  MoveAbsJ [[102.02,-14.19,-142.83,-135.95,-26.88,37.39],[9E9,9E9,9E9,9E9,9E9,9E9]],speeddata0,DefaultBlend,tool0;
  MoveAbsJ [[101.51,-13.98,-141.84,-136.12,-26.41,37.13],[9E9,9E9,9E9,9E9,9E9,9E9]],speeddata0,DefaultBlend,tool0;
  MoveAbsJ [[100.99,-13.77,-140.85,-136.29,-25.94,36.87],[9E9,9E9,9E9,9E9,9E9,9E9]],speeddata0,DefaultBlend,tool0;
  MoveAbsJ [[100.48,-13.56,-139.86,-136.46,-25.48,36.61],[9E9,9E9,9E9,9E9,9E9,9E9]],speeddata0,DefaultBlend,tool0;
  MoveAbsJ [[99.97,-13.35,-138.87,-136.62,-25.01,36.35],[9E9,9E9,9E9,9E9,9E9,9E9]],speeddata0,DefaultBlend,tool0;
  MoveAbsJ [[99.46,-13.14,-137.88,-136.79,-24.54,36.09],[9E9,9E9,9E9,9E9,9E9,9E9]],speeddata0,DefaultBlend,tool0;
  MoveAbsJ [[98.95,-12.93,-136.89,-136.96,-24.08,35.83],[9E9,9E9,9E9,9E9,9E9,9E9]],speeddata0,DefaultBlend,tool0;
  MoveAbsJ [[98.43,-12.72,-135.89,-137.13,-23.61,35.57],[9E9,9E9,9E9,9E9,9E9,9E9]],speeddata0,DefaultBlend,tool0;
  MoveAbsJ [[97.92,-12.51,-134.90,-137.29,-23.14,35.31],[9E9,9E9,9E9,9E9,9E9,9E9]],speeddata0,DefaultBlend,tool0;
  MoveAbsJ [[97.41,-12.30,-133.91,-137.46,-22.68,35.05],[9E9,9E9,9E9,9E9,9E9,9E9]],speeddata0,DefaultBlend,tool0;
  MoveAbsJ [[96.90,-12.09,-132.92,-137.63,-22.21,34.79],[9E9,9E9,9E9,9E9,9E9,9E9]],speeddata0,DefaultBlend,tool0;
  MoveAbsJ [[96.39,-11.88,-131.93,-137.80,-21.74,34.53],[9E9,9E9,9E9,9E9,9E9,9E9]],speeddata0,DefaultBlend,tool0;
  MoveAbsJ [[95.87,-11.67,-130.94,-137.97,-21.28,34.27],[9E9,9E9,9E9,9E9,9E9,9E9]],speeddata0,DefaultBlend,tool0;
  MoveAbsJ [[95.36,-11.46,-129.95,-138.13,-20.81,34.01],[9E9,9E9,9E9,9E9,9E9,9E9]],speeddata0,DefaultBlend,tool0;
  MoveAbsJ [[94.85,-11.25,-128.96,-138.30,-20.34,33.75],[9E9,9E9,9E9,9E9,9E9,9E9]],speeddata0,DefaultBlend,tool0;
  MoveAbsJ [[94.34,-11.04,-127.96,-138.47,-19.88,33.49],[9E9,9E9,9E9,9E9,9E9,9E9]],speeddata0,DefaultBlend,tool0;
  MoveAbsJ [[93.83,-10.83,-126.97,-138.64,-19.41,33.23],[9E9,9E9,9E9,9E9,9E9,9E9]],speeddata0,DefaultBlend,tool0;
  MoveAbsJ [[93.31,-10.63,-125.98,-138.80,-18.94,32.97],[9E9,9E9,9E9,9E9,9E9,9E9]],speeddata0,DefaultBlend,tool0;
  MoveAbsJ [[92.80,-10.42,-124.99,-138.97,-18.48,32.71],[9E9,9E9,9E9,9E9,9E9,9E9]],speeddata0,DefaultBlend,tool0;
  MoveAbsJ [[92.29,-10.21,-124.00,-139.14,-18.01,32.45],[9E9,9E9,9E9,9E9,9E9,9E9]],speeddata0,DefaultBlend,tool0;
  MoveAbsJ [[91.78,-10.00,-123.01,-139.31,-17.54,32.19],[9E9,9E9,9E9,9E9,9E9,9E9]],speeddata0,DefaultBlend,tool0;
  MoveAbsJ [[91.27,-9.79,-122.02,-139.47,-17.08,31.93],[9E9,9E9,9E9,9E9,9E9,9E9]],speeddata0,DefaultBlend,tool0;
  MoveAbsJ [[90.75,-9.58,-121.02,-139.64,-16.61,31.67],[9E9,9E9,9E9,9E9,9E9,9E9]],speeddata0,DefaultBlend,tool0;
  MoveAbsJ [[90.24,-9.37,-120.03,-139.81,-16.14,31.41],[9E9,9E9,9E9,9E9,9E9,9E9]],speeddata0,DefaultBlend,tool0;
  MoveAbsJ [[89.73,-9.16,-119.04,-139.98,-15.68,31.15],[9E9,9E9,9E9,9E9,9E9,9E9]],speeddata0,DefaultBlend,tool0;
  MoveAbsJ [[89.22,-8.95,-118.05,-140.14,-15.21,30.89],[9E9,9E9,9E9,9E9,9E9,9E9]],speeddata0,DefaultBlend,tool0;
  MoveAbsJ [[88.71,-8.74,-117.06,-140.31,-14.74,30.63],[9E9,9E9,9E9,9E9,9E9,9E9]],speeddata0,DefaultBlend,tool0;
  MoveAbsJ [[88.19,-8.53,-116.07,-140.48,-14.28,30.36],[9E9,9E9,9E9,9E9,9E9,9E9]],speeddata0,DefaultBlend,tool0;
  MoveAbsJ [[87.68,-8.32,-115.08,-140.65,-13.81,30.10],[9E9,9E9,9E9,9E9,9E9,9E9]],speeddata0,DefaultBlend,tool0;
  MoveAbsJ [[87.17,-8.11,-114.08,-140.82,-13.34,29.84],[9E9,9E9,9E9,9E9,9E9,9E9]],speeddata0,DefaultBlend,tool0;
  MoveAbsJ [[86.66,-7.90,-113.09,-140.98,-12.88,29.58],[9E9,9E9,9E9,9E9,9E9,9E9]],speeddata0,DefaultBlend,tool0;
  MoveAbsJ [[86.15,-7.69,-112.10,-141.15,-12.41,29.32],[9E9,9E9,9E9,9E9,9E9,9E9]],speeddata0,DefaultBlend,tool0;
  MoveAbsJ [[85.63,-7.48,-111.11,-141.32,-11.94,29.06],[9E9,9E9,9E9,9E9,9E9,9E9]],speeddata0,DefaultBlend,tool0;
  MoveAbsJ [[85.12,-7.27,-110.12,-141.49,-11.48,28.80],[9E9,9E9,9E9,9E9,9E9,9E9]],speeddata0,DefaultBlend,tool0;
  MoveAbsJ [[84.61,-7.06,-109.13,-141.65,-11.01,28.54],[9E9,9E9,9E9,9E9,9E9,9E9]],speeddata0,DefaultBlend,tool0;
  MoveAbsJ [[84.10,-6.85,-108.14,-141.82,-10.54,28.28],[9E9,9E9,9E9,9E9,9E9,9E9]],speeddata0,DefaultBlend,tool0;
  MoveAbsJ [[83.59,-6.64,-107.15,-141.99,-10.08,28.02],[9E9,9E9,9E9,9E9,9E9,9E9]],speeddata0,DefaultBlend,tool0;
  MoveAbsJ [[83.07,-6.43,-106.15,-142.16,-9.61,27.76],[9E9,9E9,9E9,9E9,9E9,9E9]],speeddata0,DefaultBlend,tool0;
  MoveAbsJ [[82.56,-6.22,-105.16,-142.32,-9.14,27.50],[9E9,9E9,9E9,9E9,9E9,9E9]],speeddata0,DefaultBlend,tool0;
  MoveAbsJ [[82.05,-6.01,-104.17,-142.49,-8.68,27.24],[9E9,9E9,9E9,9E9,9E9,9E9]],speeddata0,DefaultBlend,tool0;
  MoveAbsJ [[81.54,-5.80,-103.18,-142.66,-8.21,26.98],[9E9,9E9,9E9,9E9,9E9,9E9]],speeddata0,DefaultBlend,tool0;
  MoveAbsJ [[81.03,-5.59,-102.19,-142.83,-7.74,26.72],[9E9,9E9,9E9,9E9,9E9,9E9]],speeddata0,DefaultBlend,tool0;
  MoveAbsJ [[80.51,-5.38,-101.20,-142.99,-7.28,26.46],[9E9,9E9,9E9,9E9,9E9,9E9]],speeddata0,DefaultBlend,tool0;
  MoveAbsJ [[80.00,-5.17,-100.21,-143.16,-6.81,26.20],[9E9,9E9,9E9,9E9,9E9,9E9]],speeddata0,DefaultBlend,tool0;
  MoveAbsJ [[79.49,-4.96,-99.21,-143.33,-6.34,25.94],[9E9,9E9,9E9,9E9,9E9,9E9]],speeddata0,DefaultBlend,tool0;
  MoveAbsJ [[78.98,-4.75,-98.22,-143.50,-5.88,25.68],[9E9,9E9,9E9,9E9,9E9,9E9]],speeddata0,DefaultBlend,tool0;
  MoveAbsJ [[78.46,-4.54,-97.23,-143.67,-5.41,25.42],[9E9,9E9,9E9,9E9,9E9,9E9]],speeddata0,DefaultBlend,tool0;
  MoveAbsJ [[77.95,-4.33,-96.24,-143.83,-4.94,25.16],[9E9,9E9,9E9,9E9,9E9,9E9]],speeddata0,DefaultBlend,tool0;
  MoveAbsJ [[77.44,-4.13,-95.25,-144.00,-4.48,24.90],[9E9,9E9,9E9,9E9,9E9,9E9]],speeddata0,DefaultBlend,tool0;
  MoveAbsJ [[76.93,-3.92,-94.26,-144.17,-4.01,24.64],[9E9,9E9,9E9,9E9,9E9,9E9]],speeddata0,DefaultBlend,tool0;
  MoveAbsJ [[76.42,-3.71,-93.27,-144.34,-3.54,24.38],[9E9,9E9,9E9,9E9,9E9,9E9]],speeddata0,DefaultBlend,tool0;
  MoveAbsJ [[75.90,-3.50,-92.28,-144.50,-3.08,24.12],[9E9,9E9,9E9,9E9,9E9,9E9]],speeddata0,DefaultBlend,tool0;
  MoveAbsJ [[75.39,-3.29,-91.28,-144.67,-2.61,23.86],[9E9,9E9,9E9,9E9,9E9,9E9]],speeddata0,DefaultBlend,tool0;
  MoveAbsJ [[74.88,-3.08,-90.29,-144.84,-2.14,23.60],[9E9,9E9,9E9,9E9,9E9,9E9]],speeddata0,DefaultBlend,tool0;
  MoveAbsJ [[74.37,-2.87,-89.30,-145.01,-1.68,23.34],[9E9,9E9,9E9,9E9,9E9,9E9]],speeddata0,DefaultBlend,tool0;
  MoveAbsJ [[73.86,-2.66,-88.31,-145.17,-1.21,23.08],[9E9,9E9,9E9,9E9,9E9,9E9]],speeddata0,DefaultBlend,tool0;
  MoveAbsJ [[73.34,-2.45,-87.32,-145.34,-0.74,22.82],[9E9,9E9,9E9,9E9,9E9,9E9]],speeddata0,DefaultBlend,tool0;
  MoveAbsJ [[72.83,-2.24,-86.33,-145.51,-0.28,22.56],[9E9,9E9,9E9,9E9,9E9,9E9]],speeddata0,DefaultBlend,tool0;
  MoveAbsJ [[72.32,-2.03,-85.34,-145.68,0.19,22.30],[9E9,9E9,9E9,9E9,9E9,9E9]],speeddata0,DefaultBlend,tool0;
  MoveAbsJ [[71.81,-1.82,-84.34,-145.85,0.66,22.04],[9E9,9E9,9E9,9E9,9E9,9E9]],speeddata0,DefaultBlend,tool0;
  MoveAbsJ [[71.30,-1.61,-83.35,-146.01,1.12,21.78],[9E9,9E9,9E9,9E9,9E9,9E9]],speeddata0,DefaultBlend,tool0;
  MoveAbsJ [[70.78,-1.40,-82.36,-146.18,1.59,21.52],[9E9,9E9,9E9,9E9,9E9,9E9]],speeddata0,DefaultBlend,tool0;
  MoveAbsJ [[70.27,-1.19,-81.37,-146.35,2.06,21.26],[9E9,9E9,9E9,9E9,9E9,9E9]],speeddata0,DefaultBlend,tool0;
  MoveAbsJ [[69.76,-0.98,-80.38,-146.52,2.52,21.00],[9E9,9E9,9E9,9E9,9E9,9E9]],speeddata0,DefaultBlend,tool0;
  MoveAbsJ [[69.25,-0.77,-79.39,-146.68,2.99,20.74],[9E9,9E9,9E9,9E9,9E9,9E9]],speeddata0,DefaultBlend,tool0;
  MoveAbsJ [[68.74,-0.56,-78.40,-146.85,3.46,20.48],[9E9,9E9,9E9,9E9,9E9,9E9]],speeddata0,DefaultBlend,tool0;
  MoveAbsJ [[68.22,-0.35,-77.40,-147.02,3.92,20.22],[9E9,9E9,9E9,9E9,9E9,9E9]],speeddata0,DefaultBlend,tool0;
  MoveAbsJ [[67.71,-0.14,-76.41,-147.19,4.39,19.96],[9E9,9E9,9E9,9E9,9E9,9E9]],speeddata0,DefaultBlend,tool0;
  MoveAbsJ [[67.20,0.07,-75.42,-147.35,4.86,19.70],[9E9,9E9,9E9,9E9,9E9,9E9]],speeddata0,DefaultBlend,tool0;
  MoveAbsJ [[66.69,0.28,-74.43,-147.52,5.32,19.43],[9E9,9E9,9E9,9E9,9E9,9E9]],speeddata0,DefaultBlend,tool0;
  MoveAbsJ [[66.18,0.49,-73.44,-147.69,5.79,19.17],[9E9,9E9,9E9,9E9,9E9,9E9]],speeddata0,DefaultBlend,tool0;
  MoveAbsJ [[65.66,0.70,-72.45,-147.86,6.26,18.91],[9E9,9E9,9E9,9E9,9E9,9E9]],speeddata0,DefaultBlend,tool0;
  MoveAbsJ [[65.15,0.91,-71.46,-148.02,6.72,18.65],[9E9,9E9,9E9,9E9,9E9,9E9]],speeddata0,DefaultBlend,tool0;
  MoveAbsJ [[64.64,1.12,-70.47,-148.19,7.19,18.39],[9E9,9E9,9E9,9E9,9E9,9E9]],speeddata0,DefaultBlend,tool0;
  MoveAbsJ [[64.13,1.33,-69.47,-148.36,7.66,18.13],[9E9,9E9,9E9,9E9,9E9,9E9]],speeddata0,DefaultBlend,tool0;
  MoveAbsJ [[63.62,1.54,-68.48,-148.53,8.12,17.87],[9E9,9E9,9E9,9E9,9E9,9E9]],speeddata0,DefaultBlend,tool0;
  MoveAbsJ [[63.10,1.75,-67.49,-148.70,8.59,17.61],[9E9,9E9,9E9,9E9,9E9,9E9]],speeddata0,DefaultBlend,tool0;
  MoveAbsJ [[62.59,1.96,-66.50,-148.86,9.06,17.35],[9E9,9E9,9E9,9E9,9E9,9E9]],speeddata0,DefaultBlend,tool0;
  MoveAbsJ [[62.08,2.17,-65.51,-149.03,9.52,17.09],[9E9,9E9,9E9,9E9,9E9,9E9]],speeddata0,DefaultBlend,tool0;
  MoveAbsJ [[61.57,2.37,-64.52,-149.20,9.99,16.83],[9E9,9E9,9E9,9E9,9E9,9E9]],speeddata0,DefaultBlend,tool0;
  MoveAbsJ [[61.06,2.58,-63.53,-149.37,10.46,16.57],[9E9,9E9,9E9,9E9,9E9,9E9]],speeddata0,DefaultBlend,tool0;
  MoveAbsJ [[60.54,2.79,-62.53,-149.53,10.92,16.31],[9E9,9E9,9E9,9E9,9E9,9E9]],speeddata0,DefaultBlend,tool0;
  MoveAbsJ [[60.03,3.00,-61.54,-149.70,11.39,16.05],[9E9,9E9,9E9,9E9,9E9,9E9]],speeddata0,DefaultBlend,tool0;
  MoveAbsJ [[59.52,3.21,-60.55,-149.87,11.86,15.79],[9E9,9E9,9E9,9E9,9E9,9E9]],speeddata0,DefaultBlend,tool0;
  MoveAbsJ [[59.01,3.42,-59.56,-150.04,12.32,15.53],[9E9,9E9,9E9,9E9,9E9,9E9]],speeddata0,DefaultBlend,tool0;
  MoveAbsJ [[58.50,3.63,-58.57,-150.20,12.79,15.27],[9E9,9E9,9E9,9E9,9E9,9E9]],speeddata0,DefaultBlend,tool0;
  MoveAbsJ [[57.98,3.84,-57.58,-150.37,13.26,15.01],[9E9,9E9,9E9,9E9,9E9,9E9]],speeddata0,DefaultBlend,tool0;
  MoveAbsJ [[57.47,4.05,-56.59,-150.54,13.72,14.75],[9E9,9E9,9E9,9E9,9E9,9E9]],speeddata0,DefaultBlend,tool0;
  MoveAbsJ [[56.96,4.26,-55.59,-150.71,14.19,14.49],[9E9,9E9,9E9,9E9,9E9,9E9]],speeddata0,DefaultBlend,tool0;
  MoveAbsJ [[56.45,4.47,-54.60,-150.87,14.66,14.23],[9E9,9E9,9E9,9E9,9E9,9E9]],speeddata0,DefaultBlend,tool0;
  MoveAbsJ [[55.94,4.68,-53.61,-151.04,15.12,13.97],[9E9,9E9,9E9,9E9,9E9,9E9]],speeddata0,DefaultBlend,tool0;
  MoveAbsJ [[55.42,4.89,-52.62,-151.21,15.59,13.71],[9E9,9E9,9E9,9E9,9E9,9E9]],speeddata0,DefaultBlend,tool0;
  MoveAbsJ [[54.91,5.10,-51.63,-151.38,16.06,13.45],[9E9,9E9,9E9,9E9,9E9,9E9]],speeddata0,DefaultBlend,tool0;
  MoveAbsJ [[54.40,5.31,-50.64,-151.55,16.52,13.19],[9E9,9E9,9E9,9E9,9E9,9E9]],speeddata0,DefaultBlend,tool0;
  MoveAbsJ [[53.89,5.52,-49.65,-151.71,16.99,12.93],[9E9,9E9,9E9,9E9,9E9,9E9]],speeddata0,DefaultBlend,tool0;
  MoveAbsJ [[53.38,5.73,-48.66,-151.88,17.46,12.67],[9E9,9E9,9E9,9E9,9E9,9E9]],speeddata0,DefaultBlend,tool0;
  MoveAbsJ [[52.86,5.94,-47.66,-152.05,17.92,12.41],[9E9,9E9,9E9,9E9,9E9,9E9]],speeddata0,DefaultBlend,tool0;
  MoveAbsJ [[52.35,6.15,-46.67,-152.22,18.39,12.15],[9E9,9E9,9E9,9E9,9E9,9E9]],speeddata0,DefaultBlend,tool0;
  MoveAbsJ [[51.84,6.36,-45.68,-152.38,18.85,11.89],[9E9,9E9,9E9,9E9,9E9,9E9]],speeddata0,DefaultBlend,tool0;
  MoveAbsJ [[51.33,6.57,-44.69,-152.55,19.32,11.63],[9E9,9E9,9E9,9E9,9E9,9E9]],speeddata0,DefaultBlend,tool0;
  MoveAbsJ [[50.82,6.78,-43.70,-152.72,19.79,11.37],[9E9,9E9,9E9,9E9,9E9,9E9]],speeddata0,DefaultBlend,tool0;
  MoveAbsJ [[50.30,6.99,-42.71,-152.89,20.25,11.11],[9E9,9E9,9E9,9E9,9E9,9E9]],speeddata0,DefaultBlend,tool0;
  MoveAbsJ [[49.79,7.20,-41.72,-153.05,20.72,10.85],[9E9,9E9,9E9,9E9,9E9,9E9]],speeddata0,DefaultBlend,tool0;
  MoveAbsJ [[49.28,7.41,-40.72,-153.22,21.19,10.59],[9E9,9E9,9E9,9E9,9E9,9E9]],speeddata0,DefaultBlend,tool0;
  MoveAbsJ [[48.77,7.62,-39.73,-153.39,21.65,10.33],[9E9,9E9,9E9,9E9,9E9,9E9]],speeddata0,DefaultBlend,tool0;
  MoveAbsJ [[48.26,7.83,-38.74,-153.56,22.12,10.07],[9E9,9E9,9E9,9E9,9E9,9E9]],speeddata0,DefaultBlend,tool0;
  MoveAbsJ [[47.74,8.04,-37.75,-153.73,22.59,9.81],[9E9,9E9,9E9,9E9,9E9,9E9]],speeddata0,DefaultBlend,tool0;
  MoveAbsJ [[47.23,8.25,-36.76,-153.89,23.05,9.55],[9E9,9E9,9E9,9E9,9E9,9E9]],speeddata0,DefaultBlend,tool0;
  MoveAbsJ [[46.72,8.46,-35.77,-154.06,23.52,9.29],[9E9,9E9,9E9,9E9,9E9,9E9]],speeddata0,DefaultBlend,tool0;
  MoveAbsJ [[46.21,8.66,-34.78,-154.23,23.99,9.03],[9E9,9E9,9E9,9E9,9E9,9E9]],speeddata0,DefaultBlend,tool0;
  MoveAbsJ [[45.69,8.87,-33.79,-154.40,24.45,8.77],[9E9,9E9,9E9,9E9,9E9,9E9]],speeddata0,DefaultBlend,tool0;
  MoveAbsJ [[45.18,9.08,-32.79,-154.56,24.92,8.50],[9E9,9E9,9E9,9E9,9E9,9E9]],speeddata0,DefaultBlend,tool0;
  MoveAbsJ [[44.67,9.29,-31.80,-154.73,25.39,8.24],[9E9,9E9,9E9,9E9,9E9,9E9]],speeddata0,DefaultBlend,tool0;
  MoveAbsJ [[44.16,9.50,-30.81,-154.90,25.85,7.98],[9E9,9E9,9E9,9E9,9E9,9E9]],speeddata0,DefaultBlend,tool0;
  MoveAbsJ [[43.65,9.71,-29.82,-155.07,26.32,7.72],[9E9,9E9,9E9,9E9,9E9,9E9]],speeddata0,DefaultBlend,tool0;
  MoveAbsJ [[43.13,9.92,-28.83,-155.23,26.79,7.46],[9E9,9E9,9E9,9E9,9E9,9E9]],speeddata0,DefaultBlend,tool0;
  MoveAbsJ [[42.62,10.13,-27.84,-155.40,27.25,7.20],[9E9,9E9,9E9,9E9,9E9,9E9]],speeddata0,DefaultBlend,tool0;
  MoveAbsJ [[42.11,10.34,-26.85,-155.57,27.72,6.94],[9E9,9E9,9E9,9E9,9E9,9E9]],speeddata0,DefaultBlend,tool0;
  MoveAbsJ [[41.60,10.55,-25.85,-155.74,28.19,6.68],[9E9,9E9,9E9,9E9,9E9,9E9]],speeddata0,DefaultBlend,tool0;
  MoveAbsJ [[41.09,10.76,-24.86,-155.90,28.65,6.42],[9E9,9E9,9E9,9E9,9E9,9E9]],speeddata0,DefaultBlend,tool0;
  MoveAbsJ [[40.57,10.97,-23.87,-156.07,29.12,6.16],[9E9,9E9,9E9,9E9,9E9,9E9]],speeddata0,DefaultBlend,tool0;
  MoveAbsJ [[40.06,11.18,-22.88,-156.24,29.59,5.90],[9E9,9E9,9E9,9E9,9E9,9E9]],speeddata0,DefaultBlend,tool0;
  MoveAbsJ [[39.55,11.39,-21.89,-156.41,30.05,5.64],[9E9,9E9,9E9,9E9,9E9,9E9]],speeddata0,DefaultBlend,tool0;
  MoveAbsJ [[39.04,11.60,-20.90,-156.58,30.52,5.38],[9E9,9E9,9E9,9E9,9E9,9E9]],speeddata0,DefaultBlend,tool0;
  MoveAbsJ [[38.53,11.81,-19.91,-156.74,30.99,5.12],[9E9,9E9,9E9,9E9,9E9,9E9]],speeddata0,DefaultBlend,tool0;
  MoveAbsJ [[38.01,12.02,-18.91,-156.91,31.45,4.86],[9E9,9E9,9E9,9E9,9E9,9E9]],speeddata0,DefaultBlend,tool0;
  MoveAbsJ [[37.50,12.23,-17.92,-157.08,31.92,4.60],[9E9,9E9,9E9,9E9,9E9,9E9]],speeddata0,DefaultBlend,tool0;
  MoveAbsJ [[36.99,12.44,-16.93,-157.25,32.39,4.34],[9E9,9E9,9E9,9E9,9E9,9E9]],speeddata0,DefaultBlend,tool0;
  MoveAbsJ [[36.48,12.65,-15.94,-157.41,32.85,4.08],[9E9,9E9,9E9,9E9,9E9,9E9]],speeddata0,DefaultBlend,tool0;
  MoveAbsJ [[35.97,12.86,-14.95,-157.58,33.32,3.82],[9E9,9E9,9E9,9E9,9E9,9E9]],speeddata0,DefaultBlend,tool0;
  MoveAbsJ [[35.45,13.07,-13.96,-157.75,33.79,3.56],[9E9,9E9,9E9,9E9,9E9,9E9]],speeddata0,DefaultBlend,tool0;
  MoveAbsJ [[34.94,13.28,-12.97,-157.92,34.25,3.30],[9E9,9E9,9E9,9E9,9E9,9E9]],speeddata0,DefaultBlend,tool0;
  MoveAbsJ [[34.43,13.49,-11.98,-158.08,34.72,3.04],[9E9,9E9,9E9,9E9,9E9,9E9]],speeddata0,DefaultBlend,tool0;
  MoveAbsJ [[33.92,13.70,-10.98,-158.25,35.19,2.78],[9E9,9E9,9E9,9E9,9E9,9E9]],speeddata0,DefaultBlend,tool0;
  MoveAbsJ [[33.41,13.91,-9.99,-158.42,35.65,2.52],[9E9,9E9,9E9,9E9,9E9,9E9]],speeddata0,DefaultBlend,tool0;
  MoveAbsJ [[32.89,14.12,-9.00,-158.59,36.12,2.26],[9E9,9E9,9E9,9E9,9E9,9E9]],speeddata0,DefaultBlend,tool0;
  MoveAbsJ [[32.38,14.33,-8.01,-158.75,36.59,2.00],[9E9,9E9,9E9,9E9,9E9,9E9]],speeddata0,DefaultBlend,tool0;
  MoveAbsJ [[31.87,14.54,-7.02,-158.92,37.05,1.74],[9E9,9E9,9E9,9E9,9E9,9E9]],speeddata0,DefaultBlend,tool0;
  MoveAbsJ [[31.36,14.75,-6.03,-159.09,37.52,1.48],[9E9,9E9,9E9,9E9,9E9,9E9]],speeddata0,DefaultBlend,tool0;
  MoveAbsJ [[30.85,14.96,-5.04,-159.26,37.99,1.22],[9E9,9E9,9E9,9E9,9E9,9E9]],speeddata0,DefaultBlend,tool0;
  MoveAbsJ [[30.33,15.16,-4.04,-159.43,38.45,0.96],[9E9,9E9,9E9,9E9,9E9,9E9]],speeddata0,DefaultBlend,tool0;
  MoveAbsJ [[29.82,15.37,-3.05,-159.59,38.92,0.70],[9E9,9E9,9E9,9E9,9E9,9E9]],speeddata0,DefaultBlend,tool0;
  MoveAbsJ [[29.31,15.58,-2.06,-159.76,39.39,0.44],[9E9,9E9,9E9,9E9,9E9,9E9]],speeddata0,DefaultBlend,tool0;
  MoveAbsJ [[28.80,15.79,-1.07,-159.93,39.85,0.18],[9E9,9E9,9E9,9E9,9E9,9E9]],speeddata0,DefaultBlend,tool0;
  MoveAbsJ [[28.29,16.00,-0.08,-160.10,40.32,-0.08],[9E9,9E9,9E9,9E9,9E9,9E9]],speeddata0,DefaultBlend,tool0;
  MoveAbsJ [[27.77,16.21,0.91,-160.26,40.79,-0.34],[9E9,9E9,9E9,9E9,9E9,9E9]],speeddata0,DefaultBlend,tool0;
  MoveAbsJ [[27.26,16.42,1.90,-160.43,41.25,-0.60],[9E9,9E9,9E9,9E9,9E9,9E9]],speeddata0,DefaultBlend,tool0;
  MoveAbsJ [[26.75,16.63,2.90,-160.60,41.72,-0.86],[9E9,9E9,9E9,9E9,9E9,9E9]],speeddata0,DefaultBlend,tool0;
  MoveAbsJ [[26.24,16.84,3.89,-160.77,42.19,-1.12],[9E9,9E9,9E9,9E9,9E9,9E9]],speeddata0,DefaultBlend,tool0;
  MoveAbsJ [[25.73,17.05,4.88,-160.93,42.65,-1.38],[9E9,9E9,9E9,9E9,9E9,9E9]],speeddata0,DefaultBlend,tool0;
  MoveAbsJ [[25.21,17.26,5.87,-161.10,43.12,-1.64],[9E9,9E9,9E9,9E9,9E9,9E9]],speeddata0,DefaultBlend,tool0;
  MoveAbsJ [[24.70,17.47,6.86,-161.27,43.59,-1.90],[9E9,9E9,9E9,9E9,9E9,9E9]],speeddata0,DefaultBlend,tool0;
  MoveAbsJ [[24.19,17.68,7.85,-161.44,44.05,-2.16],[9E9,9E9,9E9,9E9,9E9,9E9]],speeddata0,DefaultBlend,tool0;
  MoveAbsJ [[23.68,17.89,8.84,-161.60,44.52,-2.42],[9E9,9E9,9E9,9E9,9E9,9E9]],speeddata0,DefaultBlend,tool0;
  MoveAbsJ [[23.17,18.10,9.83,-161.77,44.99,-2.69],[9E9,9E9,9E9,9E9,9E9,9E9]],speeddata0,DefaultBlend,tool0;
  MoveAbsJ [[22.65,18.31,10.83,-161.94,45.45,-2.95],[9E9,9E9,9E9,9E9,9E9,9E9]],speeddata0,DefaultBlend,tool0;
  MoveAbsJ [[22.14,18.52,11.82,-162.11,45.92,-3.21],[9E9,9E9,9E9,9E9,9E9,9E9]],speeddata0,DefaultBlend,tool0;
  MoveAbsJ [[21.63,18.73,12.81,-162.28,46.39,-3.47],[9E9,9E9,9E9,9E9,9E9,9E9]],speeddata0,DefaultBlend,tool0;
  MoveAbsJ [[21.12,18.94,13.80,-162.44,46.85,-3.73],[9E9,9E9,9E9,9E9,9E9,9E9]],speeddata0,DefaultBlend,tool0;
  MoveAbsJ [[20.61,19.15,14.79,-162.61,47.32,-3.99],[9E9,9E9,9E9,9E9,9E9,9E9]],speeddata0,DefaultBlend,tool0;
  MoveAbsJ [[20.09,19.36,15.78,-162.78,47.79,-4.25],[9E9,9E9,9E9,9E9,9E9,9E9]],speeddata0,DefaultBlend,tool0;
  MoveAbsJ [[19.58,19.57,16.77,-162.95,48.25,-4.51],[9E9,9E9,9E9,9E9,9E9,9E9]],speeddata0,DefaultBlend,tool0;
  MoveAbsJ [[19.07,19.78,17.77,-163.11,48.72,-4.77],[9E9,9E9,9E9,9E9,9E9,9E9]],speeddata0,DefaultBlend,tool0;
  MoveAbsJ [[18.56,19.99,18.76,-163.28,49.19,-5.03],[9E9,9E9,9E9,9E9,9E9,9E9]],speeddata0,DefaultBlend,tool0;
  MoveAbsJ [[18.05,20.20,19.75,-163.45,49.65,-5.29],[9E9,9E9,9E9,9E9,9E9,9E9]],speeddata0,DefaultBlend,tool0;
  MoveAbsJ [[17.53,20.41,20.74,-163.62,50.12,-5.55],[9E9,9E9,9E9,9E9,9E9,9E9]],speeddata0,DefaultBlend,tool0;
  MoveAbsJ [[17.02,20.62,21.73,-163.78,50.59,-5.81],[9E9,9E9,9E9,9E9,9E9,9E9]],speeddata0,DefaultBlend,tool0;
  MoveAbsJ [[16.51,20.83,22.72,-163.95,51.05,-6.07],[9E9,9E9,9E9,9E9,9E9,9E9]],speeddata0,DefaultBlend,tool0;
  MoveAbsJ [[16.00,21.04,23.71,-164.12,51.52,-6.33],[9E9,9E9,9E9,9E9,9E9,9E9]],speeddata0,DefaultBlend,tool0;
  MoveAbsJ [[15.49,21.25,24.70,-164.29,51.99,-6.59],[9E9,9E9,9E9,9E9,9E9,9E9]],speeddata0,DefaultBlend,tool0;
  MoveAbsJ [[14.97,21.46,25.70,-164.46,52.45,-6.85],[9E9,9E9,9E9,9E9,9E9,9E9]],speeddata0,DefaultBlend,tool0;
  MoveAbsJ [[14.46,21.66,26.69,-164.62,52.92,-7.11],[9E9,9E9,9E9,9E9,9E9,9E9]],speeddata0,DefaultBlend,tool0;
  MoveAbsJ [[13.95,21.87,27.68,-164.79,53.39,-7.37],[9E9,9E9,9E9,9E9,9E9,9E9]],speeddata0,DefaultBlend,tool0;
  MoveAbsJ [[13.44,22.08,28.67,-164.96,53.85,-7.63],[9E9,9E9,9E9,9E9,9E9,9E9]],speeddata0,DefaultBlend,tool0;
  MoveAbsJ [[12.93,22.29,29.66,-165.13,54.32,-7.89],[9E9,9E9,9E9,9E9,9E9,9E9]],speeddata0,DefaultBlend,tool0;
  MoveAbsJ [[12.41,22.50,30.65,-165.29,54.79,-8.15],[9E9,9E9,9E9,9E9,9E9,9E9]],speeddata0,DefaultBlend,tool0;
  MoveAbsJ [[11.90,22.71,31.64,-165.46,55.25,-8.41],[9E9,9E9,9E9,9E9,9E9,9E9]],speeddata0,FinePoint,tool0;
  TPWrite "Action 39 LinearMovement.";
  MoveAbsJ [[11.90,22.71,31.64,-165.46,55.25,-8.41],[9E9,9E9,9E9,9E9,9E9,9E9]],speeddata0,DefaultBlend,tool0;
  MoveAbsJ [[11.88,22.74,31.53,-165.47,55.15,-8.42],[9E9,9E9,9E9,9E9,9E9,9E9]],speeddata0,DefaultBlend,tool0;
  MoveAbsJ [[12.53,23.48,31.49,-164.82,55.92,-8.64],[9E9,9E9,9E9,9E9,9E9,9E9]],speeddata0,DefaultBlend,tool0;
  MoveAbsJ [[13.19,24.23,31.43,-164.16,56.68,-8.86],[9E9,9E9,9E9,9E9,9E9,9E9]],speeddata0,DefaultBlend,tool0;
  MoveAbsJ [[13.85,24.99,31.35,-163.51,57.44,-9.05],[9E9,9E9,9E9,9E9,9E9,9E9]],speeddata0,DefaultBlend,tool0;
  MoveAbsJ [[14.50,25.77,31.24,-162.86,58.19,-9.23],[9E9,9E9,9E9,9E9,9E9,9E9]],speeddata0,DefaultBlend,tool0;
  MoveAbsJ [[15.16,26.56,31.11,-162.23,58.92,-9.40],[9E9,9E9,9E9,9E9,9E9,9E9]],speeddata0,DefaultBlend,tool0;
  MoveAbsJ [[15.81,27.36,30.95,-161.60,59.64,-9.55],[9E9,9E9,9E9,9E9,9E9,9E9]],speeddata0,DefaultBlend,tool0;
  MoveAbsJ [[16.46,28.17,30.77,-160.97,60.34,-9.68],[9E9,9E9,9E9,9E9,9E9,9E9]],speeddata0,DefaultBlend,tool0;
  MoveAbsJ [[17.11,29.00,30.56,-160.36,61.04,-9.81],[9E9,9E9,9E9,9E9,9E9,9E9]],speeddata0,FinePoint,tool0;
  TPWrite "Action 40 OpenGripper.";
  TPWrite "Press Play to Continue";
  Stop;
  TPWrite "Action 41 LinearMovement.";
  MoveAbsJ [[17.11,29.00,30.56,-160.35,61.04,-9.81],[9E9,9E9,9E9,9E9,9E9,9E9]],speeddata0,DefaultBlend,tool0;
  MoveAbsJ [[17.41,28.20,31.87,-160.11,61.57,-9.77],[9E9,9E9,9E9,9E9,9E9,9E9]],speeddata0,DefaultBlend,tool0;
  MoveAbsJ [[17.72,27.37,33.22,-159.86,62.11,-9.73],[9E9,9E9,9E9,9E9,9E9,9E9]],speeddata0,DefaultBlend,tool0;
  MoveAbsJ [[18.04,26.54,34.56,-159.60,62.65,-9.70],[9E9,9E9,9E9,9E9,9E9,9E9]],speeddata0,DefaultBlend,tool0;
  MoveAbsJ [[18.36,25.72,35.89,-159.33,63.17,-9.66],[9E9,9E9,9E9,9E9,9E9,9E9]],speeddata0,DefaultBlend,tool0;
  MoveAbsJ [[18.70,24.89,37.21,-159.04,63.69,-9.64],[9E9,9E9,9E9,9E9,9E9,9E9]],speeddata0,DefaultBlend,tool0;
  MoveAbsJ [[19.05,24.07,38.51,-158.74,64.20,-9.61],[9E9,9E9,9E9,9E9,9E9,9E9]],speeddata0,DefaultBlend,tool0;
  MoveAbsJ [[19.42,23.25,39.81,-158.43,64.69,-9.59],[9E9,9E9,9E9,9E9,9E9,9E9]],speeddata0,DefaultBlend,tool0;
  MoveAbsJ [[19.79,22.42,41.09,-158.10,65.18,-9.58],[9E9,9E9,9E9,9E9,9E9,9E9]],speeddata0,FinePoint,tool0;
  TPWrite "Action 42 FreeMovement.";
  MoveAbsJ [[19.79,22.42,41.09,-158.10,65.18,-9.58],[9E9,9E9,9E9,9E9,9E9,9E9]],speeddata0,DefaultBlend,tool0;
  MoveAbsJ [[19.03,22.28,41.08,-157.96,65.07,-10.57],[9E9,9E9,9E9,9E9,9E9,9E9]],speeddata0,DefaultBlend,tool0;
  MoveAbsJ [[18.26,22.13,41.07,-157.81,64.95,-11.55],[9E9,9E9,9E9,9E9,9E9,9E9]],speeddata0,DefaultBlend,tool0;
  MoveAbsJ [[17.50,21.98,41.06,-157.67,64.84,-12.54],[9E9,9E9,9E9,9E9,9E9,9E9]],speeddata0,DefaultBlend,tool0;
  MoveAbsJ [[16.73,21.83,41.05,-157.53,64.73,-13.53],[9E9,9E9,9E9,9E9,9E9,9E9]],speeddata0,DefaultBlend,tool0;
  MoveAbsJ [[15.96,21.69,41.04,-157.39,64.61,-14.51],[9E9,9E9,9E9,9E9,9E9,9E9]],speeddata0,DefaultBlend,tool0;
  MoveAbsJ [[15.20,21.54,41.03,-157.25,64.50,-15.50],[9E9,9E9,9E9,9E9,9E9,9E9]],speeddata0,DefaultBlend,tool0;
  MoveAbsJ [[14.43,21.39,41.02,-157.11,64.39,-16.49],[9E9,9E9,9E9,9E9,9E9,9E9]],speeddata0,DefaultBlend,tool0;
  MoveAbsJ [[13.67,21.24,41.01,-156.97,64.27,-17.47],[9E9,9E9,9E9,9E9,9E9,9E9]],speeddata0,DefaultBlend,tool0;
  MoveAbsJ [[12.90,21.10,41.00,-156.83,64.16,-18.46],[9E9,9E9,9E9,9E9,9E9,9E9]],speeddata0,DefaultBlend,tool0;
  MoveAbsJ [[12.14,20.95,40.99,-156.69,64.04,-19.45],[9E9,9E9,9E9,9E9,9E9,9E9]],speeddata0,DefaultBlend,tool0;
  MoveAbsJ [[11.37,20.80,40.98,-156.55,63.93,-20.44],[9E9,9E9,9E9,9E9,9E9,9E9]],speeddata0,DefaultBlend,tool0;
  MoveAbsJ [[10.60,20.65,40.97,-156.41,63.82,-21.42],[9E9,9E9,9E9,9E9,9E9,9E9]],speeddata0,DefaultBlend,tool0;
  MoveAbsJ [[9.84,20.50,40.96,-156.27,63.70,-22.41],[9E9,9E9,9E9,9E9,9E9,9E9]],speeddata0,DefaultBlend,tool0;
  MoveAbsJ [[9.07,20.36,40.95,-156.13,63.59,-23.40],[9E9,9E9,9E9,9E9,9E9,9E9]],speeddata0,DefaultBlend,tool0;
  MoveAbsJ [[8.31,20.21,40.94,-155.99,63.47,-24.38],[9E9,9E9,9E9,9E9,9E9,9E9]],speeddata0,DefaultBlend,tool0;
  MoveAbsJ [[7.54,20.06,40.93,-155.84,63.36,-25.37],[9E9,9E9,9E9,9E9,9E9,9E9]],speeddata0,DefaultBlend,tool0;
  MoveAbsJ [[6.78,19.91,40.92,-155.70,63.25,-26.36],[9E9,9E9,9E9,9E9,9E9,9E9]],speeddata0,DefaultBlend,tool0;
  MoveAbsJ [[6.01,19.77,40.91,-155.56,63.13,-27.34],[9E9,9E9,9E9,9E9,9E9,9E9]],speeddata0,DefaultBlend,tool0;
  MoveAbsJ [[5.25,19.62,40.90,-155.42,63.02,-28.33],[9E9,9E9,9E9,9E9,9E9,9E9]],speeddata0,DefaultBlend,tool0;
  MoveAbsJ [[4.48,19.47,40.89,-155.28,62.91,-29.32],[9E9,9E9,9E9,9E9,9E9,9E9]],speeddata0,DefaultBlend,tool0;
  MoveAbsJ [[3.71,19.32,40.88,-155.14,62.79,-30.31],[9E9,9E9,9E9,9E9,9E9,9E9]],speeddata0,DefaultBlend,tool0;
  MoveAbsJ [[2.95,19.18,40.87,-155.00,62.68,-31.29],[9E9,9E9,9E9,9E9,9E9,9E9]],speeddata0,DefaultBlend,tool0;
  MoveAbsJ [[2.18,19.03,40.86,-154.86,62.56,-32.28],[9E9,9E9,9E9,9E9,9E9,9E9]],speeddata0,DefaultBlend,tool0;
  MoveAbsJ [[1.42,18.88,40.85,-154.72,62.45,-33.27],[9E9,9E9,9E9,9E9,9E9,9E9]],speeddata0,DefaultBlend,tool0;
  MoveAbsJ [[0.65,18.73,40.84,-154.58,62.34,-34.25],[9E9,9E9,9E9,9E9,9E9,9E9]],speeddata0,DefaultBlend,tool0;
  MoveAbsJ [[-0.11,18.59,40.83,-154.44,62.22,-35.24],[9E9,9E9,9E9,9E9,9E9,9E9]],speeddata0,DefaultBlend,tool0;
  MoveAbsJ [[-0.88,18.44,40.83,-154.30,62.11,-36.23],[9E9,9E9,9E9,9E9,9E9,9E9]],speeddata0,DefaultBlend,tool0;
  MoveAbsJ [[-1.65,18.29,40.82,-154.16,61.99,-37.21],[9E9,9E9,9E9,9E9,9E9,9E9]],speeddata0,DefaultBlend,tool0;
  MoveAbsJ [[-2.41,18.14,40.81,-154.02,61.88,-38.20],[9E9,9E9,9E9,9E9,9E9,9E9]],speeddata0,DefaultBlend,tool0;
  MoveAbsJ [[-3.18,18.00,40.80,-153.87,61.77,-39.19],[9E9,9E9,9E9,9E9,9E9,9E9]],speeddata0,DefaultBlend,tool0;
  MoveAbsJ [[-3.94,17.85,40.79,-153.73,61.65,-40.18],[9E9,9E9,9E9,9E9,9E9,9E9]],speeddata0,DefaultBlend,tool0;
  MoveAbsJ [[-4.71,17.70,40.78,-153.59,61.54,-41.16],[9E9,9E9,9E9,9E9,9E9,9E9]],speeddata0,DefaultBlend,tool0;
  MoveAbsJ [[-5.47,17.55,40.77,-153.45,61.43,-42.15],[9E9,9E9,9E9,9E9,9E9,9E9]],speeddata0,DefaultBlend,tool0;
  MoveAbsJ [[-6.24,17.41,40.76,-153.31,61.31,-43.14],[9E9,9E9,9E9,9E9,9E9,9E9]],speeddata0,DefaultBlend,tool0;
  MoveAbsJ [[-7.01,17.26,40.75,-153.17,61.20,-44.12],[9E9,9E9,9E9,9E9,9E9,9E9]],speeddata0,DefaultBlend,tool0;
  MoveAbsJ [[-7.77,17.11,40.74,-153.03,61.08,-45.11],[9E9,9E9,9E9,9E9,9E9,9E9]],speeddata0,DefaultBlend,tool0;
  MoveAbsJ [[-8.54,16.96,40.73,-152.89,60.97,-46.10],[9E9,9E9,9E9,9E9,9E9,9E9]],speeddata0,DefaultBlend,tool0;
  MoveAbsJ [[-9.30,16.82,40.72,-152.75,60.86,-47.08],[9E9,9E9,9E9,9E9,9E9,9E9]],speeddata0,DefaultBlend,tool0;
  MoveAbsJ [[-10.07,16.67,40.71,-152.61,60.74,-48.07],[9E9,9E9,9E9,9E9,9E9,9E9]],speeddata0,DefaultBlend,tool0;
  MoveAbsJ [[-10.83,16.52,40.70,-152.47,60.63,-49.06],[9E9,9E9,9E9,9E9,9E9,9E9]],speeddata0,DefaultBlend,tool0;
  MoveAbsJ [[-11.60,16.37,40.69,-152.33,60.51,-50.05],[9E9,9E9,9E9,9E9,9E9,9E9]],speeddata0,DefaultBlend,tool0;
  MoveAbsJ [[-12.37,16.23,40.68,-152.19,60.40,-51.03],[9E9,9E9,9E9,9E9,9E9,9E9]],speeddata0,DefaultBlend,tool0;
  MoveAbsJ [[-13.13,16.08,40.67,-152.05,60.29,-52.02],[9E9,9E9,9E9,9E9,9E9,9E9]],speeddata0,DefaultBlend,tool0;
  MoveAbsJ [[-13.90,15.93,40.66,-151.90,60.17,-53.01],[9E9,9E9,9E9,9E9,9E9,9E9]],speeddata0,DefaultBlend,tool0;
  MoveAbsJ [[-14.66,15.78,40.65,-151.76,60.06,-53.99],[9E9,9E9,9E9,9E9,9E9,9E9]],speeddata0,DefaultBlend,tool0;
  MoveAbsJ [[-15.43,15.64,40.64,-151.62,59.95,-54.98],[9E9,9E9,9E9,9E9,9E9,9E9]],speeddata0,DefaultBlend,tool0;
  MoveAbsJ [[-16.19,15.49,40.63,-151.48,59.83,-55.97],[9E9,9E9,9E9,9E9,9E9,9E9]],speeddata0,DefaultBlend,tool0;
  MoveAbsJ [[-16.96,15.34,40.62,-151.34,59.72,-56.95],[9E9,9E9,9E9,9E9,9E9,9E9]],speeddata0,DefaultBlend,tool0;
  MoveAbsJ [[-17.73,15.19,40.61,-151.20,59.60,-57.94],[9E9,9E9,9E9,9E9,9E9,9E9]],speeddata0,DefaultBlend,tool0;
  MoveAbsJ [[-18.49,15.05,40.60,-151.06,59.49,-58.93],[9E9,9E9,9E9,9E9,9E9,9E9]],speeddata0,DefaultBlend,tool0;
  MoveAbsJ [[-19.26,14.90,40.59,-150.92,59.38,-59.92],[9E9,9E9,9E9,9E9,9E9,9E9]],speeddata0,DefaultBlend,tool0;
  MoveAbsJ [[-20.02,14.75,40.58,-150.78,59.26,-60.90],[9E9,9E9,9E9,9E9,9E9,9E9]],speeddata0,DefaultBlend,tool0;
  MoveAbsJ [[-20.79,14.60,40.57,-150.64,59.15,-61.89],[9E9,9E9,9E9,9E9,9E9,9E9]],speeddata0,DefaultBlend,tool0;
  MoveAbsJ [[-21.55,14.46,40.56,-150.50,59.03,-62.88],[9E9,9E9,9E9,9E9,9E9,9E9]],speeddata0,DefaultBlend,tool0;
  MoveAbsJ [[-22.32,14.31,40.56,-150.36,58.92,-63.86],[9E9,9E9,9E9,9E9,9E9,9E9]],speeddata0,DefaultBlend,tool0;
  MoveAbsJ [[-23.08,14.16,40.55,-150.22,58.81,-64.85],[9E9,9E9,9E9,9E9,9E9,9E9]],speeddata0,DefaultBlend,tool0;
  MoveAbsJ [[-23.85,14.01,40.54,-150.08,58.69,-65.84],[9E9,9E9,9E9,9E9,9E9,9E9]],speeddata0,DefaultBlend,tool0;
  MoveAbsJ [[-24.62,13.86,40.53,-149.93,58.58,-66.82],[9E9,9E9,9E9,9E9,9E9,9E9]],speeddata0,DefaultBlend,tool0;
  MoveAbsJ [[-25.38,13.72,40.52,-149.79,58.47,-67.81],[9E9,9E9,9E9,9E9,9E9,9E9]],speeddata0,DefaultBlend,tool0;
  MoveAbsJ [[-26.15,13.57,40.51,-149.65,58.35,-68.80],[9E9,9E9,9E9,9E9,9E9,9E9]],speeddata0,DefaultBlend,tool0;
  MoveAbsJ [[-26.91,13.42,40.50,-149.51,58.24,-69.79],[9E9,9E9,9E9,9E9,9E9,9E9]],speeddata0,DefaultBlend,tool0;
  MoveAbsJ [[-27.68,13.27,40.49,-149.37,58.12,-70.77],[9E9,9E9,9E9,9E9,9E9,9E9]],speeddata0,DefaultBlend,tool0;
  MoveAbsJ [[-28.44,13.13,40.48,-149.23,58.01,-71.76],[9E9,9E9,9E9,9E9,9E9,9E9]],speeddata0,DefaultBlend,tool0;
  MoveAbsJ [[-29.21,12.98,40.47,-149.09,57.90,-72.75],[9E9,9E9,9E9,9E9,9E9,9E9]],speeddata0,DefaultBlend,tool0;
  MoveAbsJ [[-29.98,12.83,40.46,-148.95,57.78,-73.73],[9E9,9E9,9E9,9E9,9E9,9E9]],speeddata0,DefaultBlend,tool0;
  MoveAbsJ [[-30.74,12.68,40.45,-148.81,57.67,-74.72],[9E9,9E9,9E9,9E9,9E9,9E9]],speeddata0,DefaultBlend,tool0;
  MoveAbsJ [[-31.51,12.54,40.44,-148.67,57.56,-75.71],[9E9,9E9,9E9,9E9,9E9,9E9]],speeddata0,DefaultBlend,tool0;
  MoveAbsJ [[-32.27,12.39,40.43,-148.53,57.44,-76.69],[9E9,9E9,9E9,9E9,9E9,9E9]],speeddata0,DefaultBlend,tool0;
  MoveAbsJ [[-33.04,12.24,40.42,-148.39,57.33,-77.68],[9E9,9E9,9E9,9E9,9E9,9E9]],speeddata0,DefaultBlend,tool0;
  MoveAbsJ [[-33.80,12.09,40.41,-148.25,57.21,-78.67],[9E9,9E9,9E9,9E9,9E9,9E9]],speeddata0,DefaultBlend,tool0;
  MoveAbsJ [[-34.57,11.95,40.40,-148.11,57.10,-79.66],[9E9,9E9,9E9,9E9,9E9,9E9]],speeddata0,DefaultBlend,tool0;
  MoveAbsJ [[-35.34,11.80,40.39,-147.96,56.99,-80.64],[9E9,9E9,9E9,9E9,9E9,9E9]],speeddata0,DefaultBlend,tool0;
  MoveAbsJ [[-36.10,11.65,40.38,-147.82,56.87,-81.63],[9E9,9E9,9E9,9E9,9E9,9E9]],speeddata0,DefaultBlend,tool0;
  MoveAbsJ [[-36.87,11.50,40.37,-147.68,56.76,-82.62],[9E9,9E9,9E9,9E9,9E9,9E9]],speeddata0,DefaultBlend,tool0;
  MoveAbsJ [[-37.63,11.36,40.36,-147.54,56.64,-83.60],[9E9,9E9,9E9,9E9,9E9,9E9]],speeddata0,DefaultBlend,tool0;
  MoveAbsJ [[-38.40,11.21,40.35,-147.40,56.53,-84.59],[9E9,9E9,9E9,9E9,9E9,9E9]],speeddata0,DefaultBlend,tool0;
  MoveAbsJ [[-39.16,11.06,40.34,-147.26,56.42,-85.58],[9E9,9E9,9E9,9E9,9E9,9E9]],speeddata0,DefaultBlend,tool0;
  MoveAbsJ [[-39.93,10.91,40.33,-147.12,56.30,-86.56],[9E9,9E9,9E9,9E9,9E9,9E9]],speeddata0,DefaultBlend,tool0;
  MoveAbsJ [[-40.70,10.77,40.32,-146.98,56.19,-87.55],[9E9,9E9,9E9,9E9,9E9,9E9]],speeddata0,DefaultBlend,tool0;
  MoveAbsJ [[-41.46,10.62,40.31,-146.84,56.08,-88.54],[9E9,9E9,9E9,9E9,9E9,9E9]],speeddata0,DefaultBlend,tool0;
  MoveAbsJ [[-42.23,10.47,40.30,-146.70,55.96,-89.53],[9E9,9E9,9E9,9E9,9E9,9E9]],speeddata0,DefaultBlend,tool0;
  MoveAbsJ [[-42.99,10.32,40.29,-146.56,55.85,-90.51],[9E9,9E9,9E9,9E9,9E9,9E9]],speeddata0,DefaultBlend,tool0;
  MoveAbsJ [[-43.76,10.18,40.28,-146.42,55.73,-91.50],[9E9,9E9,9E9,9E9,9E9,9E9]],speeddata0,DefaultBlend,tool0;
  MoveAbsJ [[-44.52,10.03,40.28,-146.28,55.62,-92.49],[9E9,9E9,9E9,9E9,9E9,9E9]],speeddata0,DefaultBlend,tool0;
  MoveAbsJ [[-45.29,9.88,40.27,-146.14,55.51,-93.47],[9E9,9E9,9E9,9E9,9E9,9E9]],speeddata0,DefaultBlend,tool0;
  MoveAbsJ [[-46.05,9.73,40.26,-145.99,55.39,-94.46],[9E9,9E9,9E9,9E9,9E9,9E9]],speeddata0,DefaultBlend,tool0;
  MoveAbsJ [[-46.82,9.59,40.25,-145.85,55.28,-95.45],[9E9,9E9,9E9,9E9,9E9,9E9]],speeddata0,DefaultBlend,tool0;
  MoveAbsJ [[-47.59,9.44,40.24,-145.71,55.16,-96.43],[9E9,9E9,9E9,9E9,9E9,9E9]],speeddata0,DefaultBlend,tool0;
  MoveAbsJ [[-48.35,9.29,40.23,-145.57,55.05,-97.42],[9E9,9E9,9E9,9E9,9E9,9E9]],speeddata0,DefaultBlend,tool0;
  MoveAbsJ [[-49.12,9.14,40.22,-145.43,54.94,-98.41],[9E9,9E9,9E9,9E9,9E9,9E9]],speeddata0,DefaultBlend,tool0;
  MoveAbsJ [[-49.88,9.00,40.21,-145.29,54.82,-99.40],[9E9,9E9,9E9,9E9,9E9,9E9]],speeddata0,DefaultBlend,tool0;
  MoveAbsJ [[-50.65,8.85,40.20,-145.15,54.71,-100.38],[9E9,9E9,9E9,9E9,9E9,9E9]],speeddata0,DefaultBlend,tool0;
  MoveAbsJ [[-51.41,8.70,40.19,-145.01,54.60,-101.37],[9E9,9E9,9E9,9E9,9E9,9E9]],speeddata0,DefaultBlend,tool0;
  MoveAbsJ [[-52.18,8.55,40.18,-144.87,54.48,-102.36],[9E9,9E9,9E9,9E9,9E9,9E9]],speeddata0,DefaultBlend,tool0;
  MoveAbsJ [[-52.95,8.41,40.17,-144.73,54.37,-103.34],[9E9,9E9,9E9,9E9,9E9,9E9]],speeddata0,DefaultBlend,tool0;
  MoveAbsJ [[-53.71,8.26,40.16,-144.59,54.25,-104.33],[9E9,9E9,9E9,9E9,9E9,9E9]],speeddata0,DefaultBlend,tool0;
  MoveAbsJ [[-54.48,8.11,40.15,-144.45,54.14,-105.32],[9E9,9E9,9E9,9E9,9E9,9E9]],speeddata0,DefaultBlend,tool0;
  MoveAbsJ [[-55.24,7.96,40.14,-144.31,54.03,-106.30],[9E9,9E9,9E9,9E9,9E9,9E9]],speeddata0,DefaultBlend,tool0;
  MoveAbsJ [[-56.01,7.82,40.13,-144.17,53.91,-107.29],[9E9,9E9,9E9,9E9,9E9,9E9]],speeddata0,DefaultBlend,tool0;
  MoveAbsJ [[-56.77,7.67,40.12,-144.02,53.80,-108.28],[9E9,9E9,9E9,9E9,9E9,9E9]],speeddata0,DefaultBlend,tool0;
  MoveAbsJ [[-57.54,7.52,40.11,-143.88,53.68,-109.27],[9E9,9E9,9E9,9E9,9E9,9E9]],speeddata0,DefaultBlend,tool0;
  MoveAbsJ [[-58.31,7.37,40.10,-143.74,53.57,-110.25],[9E9,9E9,9E9,9E9,9E9,9E9]],speeddata0,DefaultBlend,tool0;
  MoveAbsJ [[-59.07,7.22,40.09,-143.60,53.46,-111.24],[9E9,9E9,9E9,9E9,9E9,9E9]],speeddata0,DefaultBlend,tool0;
  MoveAbsJ [[-59.84,7.08,40.08,-143.46,53.34,-112.23],[9E9,9E9,9E9,9E9,9E9,9E9]],speeddata0,DefaultBlend,tool0;
  MoveAbsJ [[-60.60,6.93,40.07,-143.32,53.23,-113.21],[9E9,9E9,9E9,9E9,9E9,9E9]],speeddata0,DefaultBlend,tool0;
  MoveAbsJ [[-61.37,6.78,40.06,-143.18,53.12,-114.20],[9E9,9E9,9E9,9E9,9E9,9E9]],speeddata0,FinePoint,tool0;
  TPWrite "Action 43 LoadWorkpiece.";
  TPWrite "Press Play to Continue";
  Stop;
  TPWrite "Action 44 CloseGripper.";
  TPWrite "Press Play to Continue";
  Stop;
  TPWrite "Action 45 FreeMovement.";
  MoveAbsJ [[-61.37,6.78,40.06,-143.18,53.12,-114.20],[9E9,9E9,9E9,9E9,9E9,9E9]],speeddata0,DefaultBlend,tool0;
  MoveAbsJ [[-61.21,6.91,39.89,-142.19,53.39,-113.44],[9E9,9E9,9E9,9E9,9E9,9E9]],speeddata0,DefaultBlend,tool0;
  MoveAbsJ [[-61.06,7.03,39.71,-141.19,53.66,-112.68],[9E9,9E9,9E9,9E9,9E9,9E9]],speeddata0,DefaultBlend,tool0;
  MoveAbsJ [[-60.91,7.16,39.53,-140.20,53.93,-111.92],[9E9,9E9,9E9,9E9,9E9,9E9]],speeddata0,DefaultBlend,tool0;
  MoveAbsJ [[-60.75,7.28,39.36,-139.20,54.21,-111.16],[9E9,9E9,9E9,9E9,9E9,9E9]],speeddata0,DefaultBlend,tool0;
  MoveAbsJ [[-60.60,7.41,39.18,-138.21,54.48,-110.40],[9E9,9E9,9E9,9E9,9E9,9E9]],speeddata0,DefaultBlend,tool0;
  MoveAbsJ [[-60.45,7.54,39.01,-137.21,54.75,-109.64],[9E9,9E9,9E9,9E9,9E9,9E9]],speeddata0,DefaultBlend,tool0;
  MoveAbsJ [[-60.29,7.66,38.83,-136.22,55.03,-108.88],[9E9,9E9,9E9,9E9,9E9,9E9]],speeddata0,DefaultBlend,tool0;
  MoveAbsJ [[-60.14,7.79,38.65,-135.22,55.30,-108.12],[9E9,9E9,9E9,9E9,9E9,9E9]],speeddata0,DefaultBlend,tool0;
  MoveAbsJ [[-59.98,7.91,38.48,-134.23,55.57,-107.36],[9E9,9E9,9E9,9E9,9E9,9E9]],speeddata0,DefaultBlend,tool0;
  MoveAbsJ [[-59.83,8.04,38.30,-133.23,55.85,-106.60],[9E9,9E9,9E9,9E9,9E9,9E9]],speeddata0,DefaultBlend,tool0;
  MoveAbsJ [[-59.68,8.16,38.13,-132.24,56.12,-105.84],[9E9,9E9,9E9,9E9,9E9,9E9]],speeddata0,DefaultBlend,tool0;
  MoveAbsJ [[-59.52,8.29,37.95,-131.24,56.39,-105.08],[9E9,9E9,9E9,9E9,9E9,9E9]],speeddata0,DefaultBlend,tool0;
  MoveAbsJ [[-59.37,8.42,37.77,-130.25,56.66,-104.32],[9E9,9E9,9E9,9E9,9E9,9E9]],speeddata0,DefaultBlend,tool0;
  MoveAbsJ [[-59.22,8.54,37.60,-129.25,56.94,-103.56],[9E9,9E9,9E9,9E9,9E9,9E9]],speeddata0,DefaultBlend,tool0;
  MoveAbsJ [[-59.06,8.67,37.42,-128.26,57.21,-102.81],[9E9,9E9,9E9,9E9,9E9,9E9]],speeddata0,DefaultBlend,tool0;
  MoveAbsJ [[-58.91,8.79,37.25,-127.26,57.48,-102.05],[9E9,9E9,9E9,9E9,9E9,9E9]],speeddata0,DefaultBlend,tool0;
  MoveAbsJ [[-58.75,8.92,37.07,-126.27,57.76,-101.29],[9E9,9E9,9E9,9E9,9E9,9E9]],speeddata0,DefaultBlend,tool0;
  MoveAbsJ [[-58.60,9.04,36.89,-125.27,58.03,-100.53],[9E9,9E9,9E9,9E9,9E9,9E9]],speeddata0,DefaultBlend,tool0;
  MoveAbsJ [[-58.45,9.17,36.72,-124.28,58.30,-99.77],[9E9,9E9,9E9,9E9,9E9,9E9]],speeddata0,DefaultBlend,tool0;
  MoveAbsJ [[-58.29,9.29,36.54,-123.28,58.57,-99.01],[9E9,9E9,9E9,9E9,9E9,9E9]],speeddata0,DefaultBlend,tool0;
  MoveAbsJ [[-58.14,9.42,36.37,-122.29,58.85,-98.25],[9E9,9E9,9E9,9E9,9E9,9E9]],speeddata0,DefaultBlend,tool0;
  MoveAbsJ [[-57.99,9.55,36.19,-121.30,59.12,-97.49],[9E9,9E9,9E9,9E9,9E9,9E9]],speeddata0,DefaultBlend,tool0;
  MoveAbsJ [[-57.83,9.67,36.01,-120.30,59.39,-96.73],[9E9,9E9,9E9,9E9,9E9,9E9]],speeddata0,DefaultBlend,tool0;
  MoveAbsJ [[-57.68,9.80,35.84,-119.31,59.67,-95.97],[9E9,9E9,9E9,9E9,9E9,9E9]],speeddata0,DefaultBlend,tool0;
  MoveAbsJ [[-57.52,9.92,35.66,-118.31,59.94,-95.21],[9E9,9E9,9E9,9E9,9E9,9E9]],speeddata0,DefaultBlend,tool0;
  MoveAbsJ [[-57.37,10.05,35.49,-117.32,60.21,-94.45],[9E9,9E9,9E9,9E9,9E9,9E9]],speeddata0,DefaultBlend,tool0;
  MoveAbsJ [[-57.22,10.17,35.31,-116.32,60.49,-93.69],[9E9,9E9,9E9,9E9,9E9,9E9]],speeddata0,DefaultBlend,tool0;
  MoveAbsJ [[-57.06,10.30,35.13,-115.33,60.76,-92.93],[9E9,9E9,9E9,9E9,9E9,9E9]],speeddata0,DefaultBlend,tool0;
  MoveAbsJ [[-56.91,10.43,34.96,-114.33,61.03,-92.17],[9E9,9E9,9E9,9E9,9E9,9E9]],speeddata0,DefaultBlend,tool0;
  MoveAbsJ [[-56.75,10.55,34.78,-113.34,61.30,-91.41],[9E9,9E9,9E9,9E9,9E9,9E9]],speeddata0,DefaultBlend,tool0;
  MoveAbsJ [[-56.60,10.68,34.61,-112.34,61.58,-90.65],[9E9,9E9,9E9,9E9,9E9,9E9]],speeddata0,DefaultBlend,tool0;
  MoveAbsJ [[-56.45,10.80,34.43,-111.35,61.85,-89.89],[9E9,9E9,9E9,9E9,9E9,9E9]],speeddata0,DefaultBlend,tool0;
  MoveAbsJ [[-56.29,10.93,34.25,-110.35,62.12,-89.13],[9E9,9E9,9E9,9E9,9E9,9E9]],speeddata0,DefaultBlend,tool0;
  MoveAbsJ [[-56.14,11.05,34.08,-109.36,62.40,-88.37],[9E9,9E9,9E9,9E9,9E9,9E9]],speeddata0,DefaultBlend,tool0;
  MoveAbsJ [[-55.99,11.18,33.90,-108.36,62.67,-87.61],[9E9,9E9,9E9,9E9,9E9,9E9]],speeddata0,DefaultBlend,tool0;
  MoveAbsJ [[-55.83,11.30,33.73,-107.37,62.94,-86.85],[9E9,9E9,9E9,9E9,9E9,9E9]],speeddata0,DefaultBlend,tool0;
  MoveAbsJ [[-55.68,11.43,33.55,-106.37,63.21,-86.09],[9E9,9E9,9E9,9E9,9E9,9E9]],speeddata0,DefaultBlend,tool0;
  MoveAbsJ [[-55.52,11.56,33.37,-105.38,63.49,-85.33],[9E9,9E9,9E9,9E9,9E9,9E9]],speeddata0,DefaultBlend,tool0;
  MoveAbsJ [[-55.37,11.68,33.20,-104.38,63.76,-84.57],[9E9,9E9,9E9,9E9,9E9,9E9]],speeddata0,DefaultBlend,tool0;
  MoveAbsJ [[-55.22,11.81,33.02,-103.39,64.03,-83.81],[9E9,9E9,9E9,9E9,9E9,9E9]],speeddata0,DefaultBlend,tool0;
  MoveAbsJ [[-55.06,11.93,32.85,-102.39,64.31,-83.05],[9E9,9E9,9E9,9E9,9E9,9E9]],speeddata0,DefaultBlend,tool0;
  MoveAbsJ [[-54.91,12.06,32.67,-101.40,64.58,-82.29],[9E9,9E9,9E9,9E9,9E9,9E9]],speeddata0,DefaultBlend,tool0;
  MoveAbsJ [[-54.76,12.18,32.49,-100.41,64.85,-81.53],[9E9,9E9,9E9,9E9,9E9,9E9]],speeddata0,DefaultBlend,tool0;
  MoveAbsJ [[-54.60,12.31,32.32,-99.41,65.13,-80.78],[9E9,9E9,9E9,9E9,9E9,9E9]],speeddata0,DefaultBlend,tool0;
  MoveAbsJ [[-54.45,12.44,32.14,-98.42,65.40,-80.02],[9E9,9E9,9E9,9E9,9E9,9E9]],speeddata0,DefaultBlend,tool0;
  MoveAbsJ [[-54.29,12.56,31.96,-97.42,65.67,-79.26],[9E9,9E9,9E9,9E9,9E9,9E9]],speeddata0,DefaultBlend,tool0;
  MoveAbsJ [[-54.14,12.69,31.79,-96.43,65.94,-78.50],[9E9,9E9,9E9,9E9,9E9,9E9]],speeddata0,DefaultBlend,tool0;
  MoveAbsJ [[-53.99,12.81,31.61,-95.43,66.22,-77.74],[9E9,9E9,9E9,9E9,9E9,9E9]],speeddata0,DefaultBlend,tool0;
  MoveAbsJ [[-53.83,12.94,31.44,-94.44,66.49,-76.98],[9E9,9E9,9E9,9E9,9E9,9E9]],speeddata0,DefaultBlend,tool0;
  MoveAbsJ [[-53.68,13.06,31.26,-93.44,66.76,-76.22],[9E9,9E9,9E9,9E9,9E9,9E9]],speeddata0,DefaultBlend,tool0;
  MoveAbsJ [[-53.53,13.19,31.08,-92.45,67.04,-75.46],[9E9,9E9,9E9,9E9,9E9,9E9]],speeddata0,DefaultBlend,tool0;
  MoveAbsJ [[-53.37,13.32,30.91,-91.45,67.31,-74.70],[9E9,9E9,9E9,9E9,9E9,9E9]],speeddata0,DefaultBlend,tool0;
  MoveAbsJ [[-53.22,13.44,30.73,-90.46,67.58,-73.94],[9E9,9E9,9E9,9E9,9E9,9E9]],speeddata0,DefaultBlend,tool0;
  MoveAbsJ [[-53.06,13.57,30.56,-89.46,67.85,-73.18],[9E9,9E9,9E9,9E9,9E9,9E9]],speeddata0,DefaultBlend,tool0;
  MoveAbsJ [[-52.91,13.69,30.38,-88.47,68.13,-72.42],[9E9,9E9,9E9,9E9,9E9,9E9]],speeddata0,DefaultBlend,tool0;
  MoveAbsJ [[-52.76,13.82,30.20,-87.47,68.40,-71.66],[9E9,9E9,9E9,9E9,9E9,9E9]],speeddata0,DefaultBlend,tool0;
  MoveAbsJ [[-52.60,13.94,30.03,-86.48,68.67,-70.90],[9E9,9E9,9E9,9E9,9E9,9E9]],speeddata0,DefaultBlend,tool0;
  MoveAbsJ [[-52.45,14.07,29.85,-85.48,68.95,-70.14],[9E9,9E9,9E9,9E9,9E9,9E9]],speeddata0,DefaultBlend,tool0;
  MoveAbsJ [[-52.30,14.19,29.68,-84.49,69.22,-69.38],[9E9,9E9,9E9,9E9,9E9,9E9]],speeddata0,DefaultBlend,tool0;
  MoveAbsJ [[-52.14,14.32,29.50,-83.49,69.49,-68.62],[9E9,9E9,9E9,9E9,9E9,9E9]],speeddata0,DefaultBlend,tool0;
  MoveAbsJ [[-51.99,14.45,29.32,-82.50,69.77,-67.86],[9E9,9E9,9E9,9E9,9E9,9E9]],speeddata0,DefaultBlend,tool0;
  MoveAbsJ [[-51.83,14.57,29.15,-81.50,70.04,-67.10],[9E9,9E9,9E9,9E9,9E9,9E9]],speeddata0,DefaultBlend,tool0;
  MoveAbsJ [[-51.68,14.70,28.97,-80.51,70.31,-66.34],[9E9,9E9,9E9,9E9,9E9,9E9]],speeddata0,DefaultBlend,tool0;
  MoveAbsJ [[-51.53,14.82,28.80,-79.52,70.58,-65.58],[9E9,9E9,9E9,9E9,9E9,9E9]],speeddata0,DefaultBlend,tool0;
  MoveAbsJ [[-51.37,14.95,28.62,-78.52,70.86,-64.82],[9E9,9E9,9E9,9E9,9E9,9E9]],speeddata0,DefaultBlend,tool0;
  MoveAbsJ [[-51.22,15.07,28.44,-77.53,71.13,-64.06],[9E9,9E9,9E9,9E9,9E9,9E9]],speeddata0,DefaultBlend,tool0;
  MoveAbsJ [[-51.07,15.20,28.27,-76.53,71.40,-63.30],[9E9,9E9,9E9,9E9,9E9,9E9]],speeddata0,DefaultBlend,tool0;
  MoveAbsJ [[-50.91,15.33,28.09,-75.54,71.68,-62.54],[9E9,9E9,9E9,9E9,9E9,9E9]],speeddata0,DefaultBlend,tool0;
  MoveAbsJ [[-50.76,15.45,27.92,-74.54,71.95,-61.78],[9E9,9E9,9E9,9E9,9E9,9E9]],speeddata0,DefaultBlend,tool0;
  MoveAbsJ [[-50.60,15.58,27.74,-73.55,72.22,-61.02],[9E9,9E9,9E9,9E9,9E9,9E9]],speeddata0,DefaultBlend,tool0;
  MoveAbsJ [[-50.45,15.70,27.56,-72.55,72.49,-60.26],[9E9,9E9,9E9,9E9,9E9,9E9]],speeddata0,DefaultBlend,tool0;
  MoveAbsJ [[-50.30,15.83,27.39,-71.56,72.77,-59.50],[9E9,9E9,9E9,9E9,9E9,9E9]],speeddata0,DefaultBlend,tool0;
  MoveAbsJ [[-50.14,15.95,27.21,-70.56,73.04,-58.75],[9E9,9E9,9E9,9E9,9E9,9E9]],speeddata0,DefaultBlend,tool0;
  MoveAbsJ [[-49.99,16.08,27.04,-69.57,73.31,-57.99],[9E9,9E9,9E9,9E9,9E9,9E9]],speeddata0,DefaultBlend,tool0;
  MoveAbsJ [[-49.84,16.20,26.86,-68.57,73.59,-57.23],[9E9,9E9,9E9,9E9,9E9,9E9]],speeddata0,DefaultBlend,tool0;
  MoveAbsJ [[-49.68,16.33,26.68,-67.58,73.86,-56.47],[9E9,9E9,9E9,9E9,9E9,9E9]],speeddata0,DefaultBlend,tool0;
  MoveAbsJ [[-49.53,16.46,26.51,-66.58,74.13,-55.71],[9E9,9E9,9E9,9E9,9E9,9E9]],speeddata0,DefaultBlend,tool0;
  MoveAbsJ [[-49.37,16.58,26.33,-65.59,74.41,-54.95],[9E9,9E9,9E9,9E9,9E9,9E9]],speeddata0,DefaultBlend,tool0;
  MoveAbsJ [[-49.22,16.71,26.16,-64.59,74.68,-54.19],[9E9,9E9,9E9,9E9,9E9,9E9]],speeddata0,DefaultBlend,tool0;
  MoveAbsJ [[-49.07,16.83,25.98,-63.60,74.95,-53.43],[9E9,9E9,9E9,9E9,9E9,9E9]],speeddata0,DefaultBlend,tool0;
  MoveAbsJ [[-48.91,16.96,25.80,-62.60,75.22,-52.67],[9E9,9E9,9E9,9E9,9E9,9E9]],speeddata0,DefaultBlend,tool0;
  MoveAbsJ [[-48.76,17.08,25.63,-61.61,75.50,-51.91],[9E9,9E9,9E9,9E9,9E9,9E9]],speeddata0,DefaultBlend,tool0;
  MoveAbsJ [[-48.60,17.21,25.45,-60.61,75.77,-51.15],[9E9,9E9,9E9,9E9,9E9,9E9]],speeddata0,DefaultBlend,tool0;
  MoveAbsJ [[-48.45,17.34,25.27,-59.62,76.04,-50.39],[9E9,9E9,9E9,9E9,9E9,9E9]],speeddata0,DefaultBlend,tool0;
  MoveAbsJ [[-48.30,17.46,25.10,-58.63,76.32,-49.63],[9E9,9E9,9E9,9E9,9E9,9E9]],speeddata0,DefaultBlend,tool0;
  MoveAbsJ [[-48.14,17.59,24.92,-57.63,76.59,-48.87],[9E9,9E9,9E9,9E9,9E9,9E9]],speeddata0,DefaultBlend,tool0;
  MoveAbsJ [[-47.99,17.71,24.75,-56.64,76.86,-48.11],[9E9,9E9,9E9,9E9,9E9,9E9]],speeddata0,DefaultBlend,tool0;
  MoveAbsJ [[-47.84,17.84,24.57,-55.64,77.13,-47.35],[9E9,9E9,9E9,9E9,9E9,9E9]],speeddata0,DefaultBlend,tool0;
  MoveAbsJ [[-47.68,17.96,24.39,-54.65,77.41,-46.59],[9E9,9E9,9E9,9E9,9E9,9E9]],speeddata0,DefaultBlend,tool0;
  MoveAbsJ [[-47.53,18.09,24.22,-53.65,77.68,-45.83],[9E9,9E9,9E9,9E9,9E9,9E9]],speeddata0,DefaultBlend,tool0;
  MoveAbsJ [[-47.37,18.21,24.04,-52.66,77.95,-45.07],[9E9,9E9,9E9,9E9,9E9,9E9]],speeddata0,DefaultBlend,tool0;
  MoveAbsJ [[-47.22,18.34,23.87,-51.66,78.23,-44.31],[9E9,9E9,9E9,9E9,9E9,9E9]],speeddata0,DefaultBlend,tool0;
  MoveAbsJ [[-47.07,18.47,23.69,-50.67,78.50,-43.55],[9E9,9E9,9E9,9E9,9E9,9E9]],speeddata0,DefaultBlend,tool0;
  MoveAbsJ [[-46.91,18.59,23.51,-49.67,78.77,-42.79],[9E9,9E9,9E9,9E9,9E9,9E9]],speeddata0,DefaultBlend,tool0;
  MoveAbsJ [[-46.76,18.72,23.34,-48.68,79.05,-42.03],[9E9,9E9,9E9,9E9,9E9,9E9]],speeddata0,DefaultBlend,tool0;
  MoveAbsJ [[-46.61,18.84,23.16,-47.68,79.32,-41.27],[9E9,9E9,9E9,9E9,9E9,9E9]],speeddata0,DefaultBlend,tool0;
  MoveAbsJ [[-46.45,18.97,22.99,-46.69,79.59,-40.51],[9E9,9E9,9E9,9E9,9E9,9E9]],speeddata0,DefaultBlend,tool0;
  MoveAbsJ [[-46.30,19.09,22.81,-45.69,79.86,-39.75],[9E9,9E9,9E9,9E9,9E9,9E9]],speeddata0,DefaultBlend,tool0;
  MoveAbsJ [[-46.14,19.22,22.63,-44.70,80.14,-38.99],[9E9,9E9,9E9,9E9,9E9,9E9]],speeddata0,DefaultBlend,tool0;
  MoveAbsJ [[-45.99,19.35,22.46,-43.70,80.41,-38.23],[9E9,9E9,9E9,9E9,9E9,9E9]],speeddata0,DefaultBlend,tool0;
  MoveAbsJ [[-45.84,19.47,22.28,-42.71,80.68,-37.47],[9E9,9E9,9E9,9E9,9E9,9E9]],speeddata0,DefaultBlend,tool0;
  MoveAbsJ [[-45.68,19.60,22.11,-41.71,80.96,-36.71],[9E9,9E9,9E9,9E9,9E9,9E9]],speeddata0,DefaultBlend,tool0;
  MoveAbsJ [[-45.53,19.72,21.93,-40.72,81.23,-35.96],[9E9,9E9,9E9,9E9,9E9,9E9]],speeddata0,DefaultBlend,tool0;
  MoveAbsJ [[-45.38,19.85,21.75,-39.72,81.50,-35.20],[9E9,9E9,9E9,9E9,9E9,9E9]],speeddata0,DefaultBlend,tool0;
  MoveAbsJ [[-45.22,19.97,21.58,-38.73,81.77,-34.44],[9E9,9E9,9E9,9E9,9E9,9E9]],speeddata0,DefaultBlend,tool0;
  MoveAbsJ [[-45.07,20.10,21.40,-37.74,82.05,-33.68],[9E9,9E9,9E9,9E9,9E9,9E9]],speeddata0,DefaultBlend,tool0;
  MoveAbsJ [[-44.91,20.22,21.23,-36.74,82.32,-32.92],[9E9,9E9,9E9,9E9,9E9,9E9]],speeddata0,DefaultBlend,tool0;
  MoveAbsJ [[-44.76,20.35,21.05,-35.75,82.59,-32.16],[9E9,9E9,9E9,9E9,9E9,9E9]],speeddata0,DefaultBlend,tool0;
  MoveAbsJ [[-44.61,20.48,20.87,-34.75,82.87,-31.40],[9E9,9E9,9E9,9E9,9E9,9E9]],speeddata0,DefaultBlend,tool0;
  MoveAbsJ [[-44.45,20.60,20.70,-33.76,83.14,-30.64],[9E9,9E9,9E9,9E9,9E9,9E9]],speeddata0,DefaultBlend,tool0;
  MoveAbsJ [[-44.30,20.73,20.52,-32.76,83.41,-29.88],[9E9,9E9,9E9,9E9,9E9,9E9]],speeddata0,DefaultBlend,tool0;
  MoveAbsJ [[-44.15,20.85,20.35,-31.77,83.69,-29.12],[9E9,9E9,9E9,9E9,9E9,9E9]],speeddata0,DefaultBlend,tool0;
  MoveAbsJ [[-43.99,20.98,20.17,-30.77,83.96,-28.36],[9E9,9E9,9E9,9E9,9E9,9E9]],speeddata0,DefaultBlend,tool0;
  MoveAbsJ [[-43.84,21.10,19.99,-29.78,84.23,-27.60],[9E9,9E9,9E9,9E9,9E9,9E9]],speeddata0,DefaultBlend,tool0;
  MoveAbsJ [[-43.68,21.23,19.82,-28.78,84.50,-26.84],[9E9,9E9,9E9,9E9,9E9,9E9]],speeddata0,DefaultBlend,tool0;
  MoveAbsJ [[-43.53,21.36,19.64,-27.79,84.78,-26.08],[9E9,9E9,9E9,9E9,9E9,9E9]],speeddata0,DefaultBlend,tool0;
  MoveAbsJ [[-43.38,21.48,19.47,-26.79,85.05,-25.32],[9E9,9E9,9E9,9E9,9E9,9E9]],speeddata0,DefaultBlend,tool0;
  MoveAbsJ [[-43.22,21.61,19.29,-25.80,85.32,-24.56],[9E9,9E9,9E9,9E9,9E9,9E9]],speeddata0,DefaultBlend,tool0;
  MoveAbsJ [[-43.07,21.73,19.11,-24.80,85.60,-23.80],[9E9,9E9,9E9,9E9,9E9,9E9]],speeddata0,DefaultBlend,tool0;
  MoveAbsJ [[-42.92,21.86,18.94,-23.81,85.87,-23.04],[9E9,9E9,9E9,9E9,9E9,9E9]],speeddata0,DefaultBlend,tool0;
  MoveAbsJ [[-42.76,21.98,18.76,-22.81,86.14,-22.28],[9E9,9E9,9E9,9E9,9E9,9E9]],speeddata0,DefaultBlend,tool0;
  MoveAbsJ [[-42.61,22.11,18.59,-21.82,86.41,-21.52],[9E9,9E9,9E9,9E9,9E9,9E9]],speeddata0,DefaultBlend,tool0;
  MoveAbsJ [[-42.45,22.23,18.41,-20.82,86.69,-20.76],[9E9,9E9,9E9,9E9,9E9,9E9]],speeddata0,DefaultBlend,tool0;
  MoveAbsJ [[-42.30,22.36,18.23,-19.83,86.96,-20.00],[9E9,9E9,9E9,9E9,9E9,9E9]],speeddata0,DefaultBlend,tool0;
  MoveAbsJ [[-42.15,22.49,18.06,-18.83,87.23,-19.24],[9E9,9E9,9E9,9E9,9E9,9E9]],speeddata0,DefaultBlend,tool0;
  MoveAbsJ [[-41.99,22.61,17.88,-17.84,87.51,-18.48],[9E9,9E9,9E9,9E9,9E9,9E9]],speeddata0,DefaultBlend,tool0;
  MoveAbsJ [[-41.84,22.74,17.70,-16.85,87.78,-17.72],[9E9,9E9,9E9,9E9,9E9,9E9]],speeddata0,DefaultBlend,tool0;
  MoveAbsJ [[-41.68,22.86,17.53,-15.85,88.05,-16.96],[9E9,9E9,9E9,9E9,9E9,9E9]],speeddata0,DefaultBlend,tool0;
  MoveAbsJ [[-41.53,22.99,17.35,-14.86,88.33,-16.20],[9E9,9E9,9E9,9E9,9E9,9E9]],speeddata0,DefaultBlend,tool0;
  MoveAbsJ [[-41.38,23.11,17.18,-13.86,88.60,-15.44],[9E9,9E9,9E9,9E9,9E9,9E9]],speeddata0,DefaultBlend,tool0;
  MoveAbsJ [[-41.22,23.24,17.00,-12.87,88.87,-14.68],[9E9,9E9,9E9,9E9,9E9,9E9]],speeddata0,DefaultBlend,tool0;
  MoveAbsJ [[-41.07,23.37,16.82,-11.87,89.14,-13.93],[9E9,9E9,9E9,9E9,9E9,9E9]],speeddata0,DefaultBlend,tool0;
  MoveAbsJ [[-40.92,23.49,16.65,-10.88,89.42,-13.17],[9E9,9E9,9E9,9E9,9E9,9E9]],speeddata0,DefaultBlend,tool0;
  MoveAbsJ [[-40.76,23.62,16.47,-9.88,89.69,-12.41],[9E9,9E9,9E9,9E9,9E9,9E9]],speeddata0,DefaultBlend,tool0;
  MoveAbsJ [[-40.61,23.74,16.30,-8.89,89.96,-11.65],[9E9,9E9,9E9,9E9,9E9,9E9]],speeddata0,DefaultBlend,tool0;
  MoveAbsJ [[-40.45,23.87,16.12,-7.89,90.24,-10.89],[9E9,9E9,9E9,9E9,9E9,9E9]],speeddata0,DefaultBlend,tool0;
  MoveAbsJ [[-40.30,23.99,15.94,-6.90,90.51,-10.13],[9E9,9E9,9E9,9E9,9E9,9E9]],speeddata0,DefaultBlend,tool0;
  MoveAbsJ [[-40.15,24.12,15.77,-5.90,90.78,-9.37],[9E9,9E9,9E9,9E9,9E9,9E9]],speeddata0,DefaultBlend,tool0;
  MoveAbsJ [[-39.99,24.25,15.59,-4.91,91.05,-8.61],[9E9,9E9,9E9,9E9,9E9,9E9]],speeddata0,DefaultBlend,tool0;
  MoveAbsJ [[-39.84,24.37,15.42,-3.91,91.33,-7.85],[9E9,9E9,9E9,9E9,9E9,9E9]],speeddata0,DefaultBlend,tool0;
  MoveAbsJ [[-39.69,24.50,15.24,-2.92,91.60,-7.09],[9E9,9E9,9E9,9E9,9E9,9E9]],speeddata0,DefaultBlend,tool0;
  MoveAbsJ [[-39.53,24.62,15.06,-1.92,91.87,-6.33],[9E9,9E9,9E9,9E9,9E9,9E9]],speeddata0,DefaultBlend,tool0;
  MoveAbsJ [[-39.38,24.75,14.89,-0.93,92.15,-5.57],[9E9,9E9,9E9,9E9,9E9,9E9]],speeddata0,DefaultBlend,tool0;
  MoveAbsJ [[-39.22,24.87,14.71,0.07,92.42,-4.81],[9E9,9E9,9E9,9E9,9E9,9E9]],speeddata0,DefaultBlend,tool0;
  MoveAbsJ [[-39.07,25.00,14.54,1.06,92.69,-4.05],[9E9,9E9,9E9,9E9,9E9,9E9]],speeddata0,DefaultBlend,tool0;
  MoveAbsJ [[-38.92,25.12,14.36,2.06,92.97,-3.29],[9E9,9E9,9E9,9E9,9E9,9E9]],speeddata0,DefaultBlend,tool0;
  MoveAbsJ [[-38.76,25.25,14.18,3.05,93.24,-2.53],[9E9,9E9,9E9,9E9,9E9,9E9]],speeddata0,DefaultBlend,tool0;
  MoveAbsJ [[-38.61,25.38,14.01,4.04,93.51,-1.77],[9E9,9E9,9E9,9E9,9E9,9E9]],speeddata0,DefaultBlend,tool0;
  MoveAbsJ [[-38.46,25.50,13.83,5.04,93.78,-1.01],[9E9,9E9,9E9,9E9,9E9,9E9]],speeddata0,DefaultBlend,tool0;
  MoveAbsJ [[-38.30,25.63,13.66,6.03,94.06,-0.25],[9E9,9E9,9E9,9E9,9E9,9E9]],speeddata0,DefaultBlend,tool0;
  MoveAbsJ [[-38.15,25.75,13.48,7.03,94.33,0.51],[9E9,9E9,9E9,9E9,9E9,9E9]],speeddata0,DefaultBlend,tool0;
  MoveAbsJ [[-37.99,25.88,13.30,8.02,94.60,1.27],[9E9,9E9,9E9,9E9,9E9,9E9]],speeddata0,DefaultBlend,tool0;
  MoveAbsJ [[-37.84,26.00,13.13,9.02,94.88,2.03],[9E9,9E9,9E9,9E9,9E9,9E9]],speeddata0,DefaultBlend,tool0;
  MoveAbsJ [[-37.69,26.13,12.95,10.01,95.15,2.79],[9E9,9E9,9E9,9E9,9E9,9E9]],speeddata0,DefaultBlend,tool0;
  MoveAbsJ [[-37.53,26.26,12.78,11.01,95.42,3.55],[9E9,9E9,9E9,9E9,9E9,9E9]],speeddata0,DefaultBlend,tool0;
  MoveAbsJ [[-37.38,26.38,12.60,12.00,95.69,4.31],[9E9,9E9,9E9,9E9,9E9,9E9]],speeddata0,DefaultBlend,tool0;
  MoveAbsJ [[-37.23,26.51,12.42,13.00,95.97,5.07],[9E9,9E9,9E9,9E9,9E9,9E9]],speeddata0,DefaultBlend,tool0;
  MoveAbsJ [[-37.07,26.63,12.25,13.99,96.24,5.83],[9E9,9E9,9E9,9E9,9E9,9E9]],speeddata0,DefaultBlend,tool0;
  MoveAbsJ [[-36.92,26.76,12.07,14.99,96.51,6.59],[9E9,9E9,9E9,9E9,9E9,9E9]],speeddata0,DefaultBlend,tool0;
  MoveAbsJ [[-36.76,26.88,11.90,15.98,96.79,7.35],[9E9,9E9,9E9,9E9,9E9,9E9]],speeddata0,DefaultBlend,tool0;
  MoveAbsJ [[-36.61,27.01,11.72,16.98,97.06,8.11],[9E9,9E9,9E9,9E9,9E9,9E9]],speeddata0,DefaultBlend,tool0;
  MoveAbsJ [[-36.46,27.13,11.54,17.97,97.33,8.86],[9E9,9E9,9E9,9E9,9E9,9E9]],speeddata0,DefaultBlend,tool0;
  MoveAbsJ [[-36.30,27.26,11.37,18.97,97.61,9.62],[9E9,9E9,9E9,9E9,9E9,9E9]],speeddata0,DefaultBlend,tool0;
  MoveAbsJ [[-36.15,27.39,11.19,19.96,97.88,10.38],[9E9,9E9,9E9,9E9,9E9,9E9]],speeddata0,DefaultBlend,tool0;
  MoveAbsJ [[-36.00,27.51,11.02,20.96,98.15,11.14],[9E9,9E9,9E9,9E9,9E9,9E9]],speeddata0,DefaultBlend,tool0;
  MoveAbsJ [[-35.84,27.64,10.84,21.95,98.42,11.90],[9E9,9E9,9E9,9E9,9E9,9E9]],speeddata0,DefaultBlend,tool0;
  MoveAbsJ [[-35.69,27.76,10.66,22.95,98.70,12.66],[9E9,9E9,9E9,9E9,9E9,9E9]],speeddata0,DefaultBlend,tool0;
  MoveAbsJ [[-35.53,27.89,10.49,23.94,98.97,13.42],[9E9,9E9,9E9,9E9,9E9,9E9]],speeddata0,DefaultBlend,tool0;
  MoveAbsJ [[-35.38,28.01,10.31,24.93,99.24,14.18],[9E9,9E9,9E9,9E9,9E9,9E9]],speeddata0,DefaultBlend,tool0;
  MoveAbsJ [[-35.23,28.14,10.13,25.93,99.52,14.94],[9E9,9E9,9E9,9E9,9E9,9E9]],speeddata0,DefaultBlend,tool0;
  MoveAbsJ [[-35.07,28.27,9.96,26.92,99.79,15.70],[9E9,9E9,9E9,9E9,9E9,9E9]],speeddata0,DefaultBlend,tool0;
  MoveAbsJ [[-34.92,28.39,9.78,27.92,100.06,16.46],[9E9,9E9,9E9,9E9,9E9,9E9]],speeddata0,DefaultBlend,tool0;
  MoveAbsJ [[-34.76,28.52,9.61,28.91,100.33,17.22],[9E9,9E9,9E9,9E9,9E9,9E9]],speeddata0,DefaultBlend,tool0;
  MoveAbsJ [[-34.61,28.64,9.43,29.91,100.61,17.98],[9E9,9E9,9E9,9E9,9E9,9E9]],speeddata0,DefaultBlend,tool0;
  MoveAbsJ [[-34.46,28.77,9.25,30.90,100.88,18.74],[9E9,9E9,9E9,9E9,9E9,9E9]],speeddata0,DefaultBlend,tool0;
  MoveAbsJ [[-34.30,28.89,9.08,31.90,101.15,19.50],[9E9,9E9,9E9,9E9,9E9,9E9]],speeddata0,DefaultBlend,tool0;
  MoveAbsJ [[-34.15,29.02,8.90,32.89,101.43,20.26],[9E9,9E9,9E9,9E9,9E9,9E9]],speeddata0,DefaultBlend,tool0;
  MoveAbsJ [[-34.00,29.14,8.73,33.89,101.70,21.02],[9E9,9E9,9E9,9E9,9E9,9E9]],speeddata0,DefaultBlend,tool0;
  MoveAbsJ [[-33.84,29.27,8.55,34.88,101.97,21.78],[9E9,9E9,9E9,9E9,9E9,9E9]],speeddata0,DefaultBlend,tool0;
  MoveAbsJ [[-33.69,29.40,8.37,35.88,102.25,22.54],[9E9,9E9,9E9,9E9,9E9,9E9]],speeddata0,DefaultBlend,tool0;
  MoveAbsJ [[-33.53,29.52,8.20,36.87,102.52,23.30],[9E9,9E9,9E9,9E9,9E9,9E9]],speeddata0,DefaultBlend,tool0;
  MoveAbsJ [[-33.38,29.65,8.02,37.87,102.79,24.06],[9E9,9E9,9E9,9E9,9E9,9E9]],speeddata0,DefaultBlend,tool0;
  MoveAbsJ [[-33.23,29.77,7.85,38.86,103.06,24.82],[9E9,9E9,9E9,9E9,9E9,9E9]],speeddata0,DefaultBlend,tool0;
  MoveAbsJ [[-33.07,29.90,7.67,39.86,103.34,25.58],[9E9,9E9,9E9,9E9,9E9,9E9]],speeddata0,DefaultBlend,tool0;
  MoveAbsJ [[-32.92,30.02,7.49,40.85,103.61,26.34],[9E9,9E9,9E9,9E9,9E9,9E9]],speeddata0,DefaultBlend,tool0;
  MoveAbsJ [[-32.77,30.15,7.32,41.85,103.88,27.10],[9E9,9E9,9E9,9E9,9E9,9E9]],speeddata0,DefaultBlend,tool0;
  MoveAbsJ [[-32.61,30.28,7.14,42.84,104.16,27.86],[9E9,9E9,9E9,9E9,9E9,9E9]],speeddata0,DefaultBlend,tool0;
  MoveAbsJ [[-32.46,30.40,6.97,43.84,104.43,28.62],[9E9,9E9,9E9,9E9,9E9,9E9]],speeddata0,DefaultBlend,tool0;
  MoveAbsJ [[-32.30,30.53,6.79,44.83,104.70,29.38],[9E9,9E9,9E9,9E9,9E9,9E9]],speeddata0,DefaultBlend,tool0;
  MoveAbsJ [[-32.15,30.65,6.61,45.82,104.97,30.14],[9E9,9E9,9E9,9E9,9E9,9E9]],speeddata0,DefaultBlend,tool0;
  MoveAbsJ [[-32.00,30.78,6.44,46.82,105.25,30.89],[9E9,9E9,9E9,9E9,9E9,9E9]],speeddata0,DefaultBlend,tool0;
  MoveAbsJ [[-31.84,30.90,6.26,47.81,105.52,31.65],[9E9,9E9,9E9,9E9,9E9,9E9]],speeddata0,DefaultBlend,tool0;
  MoveAbsJ [[-31.69,31.03,6.09,48.81,105.79,32.41],[9E9,9E9,9E9,9E9,9E9,9E9]],speeddata0,DefaultBlend,tool0;
  MoveAbsJ [[-31.54,31.15,5.91,49.80,106.07,33.17],[9E9,9E9,9E9,9E9,9E9,9E9]],speeddata0,DefaultBlend,tool0;
  MoveAbsJ [[-31.38,31.28,5.73,50.80,106.34,33.93],[9E9,9E9,9E9,9E9,9E9,9E9]],speeddata0,DefaultBlend,tool0;
  MoveAbsJ [[-31.23,31.41,5.56,51.79,106.61,34.69],[9E9,9E9,9E9,9E9,9E9,9E9]],speeddata0,DefaultBlend,tool0;
  MoveAbsJ [[-31.07,31.53,5.38,52.79,106.89,35.45],[9E9,9E9,9E9,9E9,9E9,9E9]],speeddata0,DefaultBlend,tool0;
  MoveAbsJ [[-30.92,31.66,5.21,53.78,107.16,36.21],[9E9,9E9,9E9,9E9,9E9,9E9]],speeddata0,DefaultBlend,tool0;
  MoveAbsJ [[-30.77,31.78,5.03,54.78,107.43,36.97],[9E9,9E9,9E9,9E9,9E9,9E9]],speeddata0,DefaultBlend,tool0;
  MoveAbsJ [[-30.61,31.91,4.85,55.77,107.70,37.73],[9E9,9E9,9E9,9E9,9E9,9E9]],speeddata0,DefaultBlend,tool0;
  MoveAbsJ [[-30.46,32.03,4.68,56.77,107.98,38.49],[9E9,9E9,9E9,9E9,9E9,9E9]],speeddata0,DefaultBlend,tool0;
  MoveAbsJ [[-30.31,32.16,4.50,57.76,108.25,39.25],[9E9,9E9,9E9,9E9,9E9,9E9]],speeddata0,DefaultBlend,tool0;
  MoveAbsJ [[-30.15,32.29,4.33,58.76,108.52,40.01],[9E9,9E9,9E9,9E9,9E9,9E9]],speeddata0,DefaultBlend,tool0;
  MoveAbsJ [[-30.00,32.41,4.15,59.75,108.80,40.77],[9E9,9E9,9E9,9E9,9E9,9E9]],speeddata0,DefaultBlend,tool0;
  MoveAbsJ [[-29.84,32.54,3.97,60.75,109.07,41.53],[9E9,9E9,9E9,9E9,9E9,9E9]],speeddata0,DefaultBlend,tool0;
  MoveAbsJ [[-29.69,32.66,3.80,61.74,109.34,42.29],[9E9,9E9,9E9,9E9,9E9,9E9]],speeddata0,DefaultBlend,tool0;
  MoveAbsJ [[-29.54,32.79,3.62,62.74,109.62,43.05],[9E9,9E9,9E9,9E9,9E9,9E9]],speeddata0,DefaultBlend,tool0;
  MoveAbsJ [[-29.38,32.91,3.45,63.73,109.89,43.81],[9E9,9E9,9E9,9E9,9E9,9E9]],speeddata0,DefaultBlend,tool0;
  MoveAbsJ [[-29.23,33.04,3.27,64.73,110.16,44.57],[9E9,9E9,9E9,9E9,9E9,9E9]],speeddata0,DefaultBlend,tool0;
  MoveAbsJ [[-29.08,33.16,3.09,65.72,110.43,45.33],[9E9,9E9,9E9,9E9,9E9,9E9]],speeddata0,DefaultBlend,tool0;
  MoveAbsJ [[-28.92,33.29,2.92,66.72,110.71,46.09],[9E9,9E9,9E9,9E9,9E9,9E9]],speeddata0,DefaultBlend,tool0;
  MoveAbsJ [[-28.77,33.42,2.74,67.71,110.98,46.85],[9E9,9E9,9E9,9E9,9E9,9E9]],speeddata0,DefaultBlend,tool0;
  MoveAbsJ [[-28.61,33.54,2.56,68.70,111.25,47.61],[9E9,9E9,9E9,9E9,9E9,9E9]],speeddata0,DefaultBlend,tool0;
  MoveAbsJ [[-28.46,33.67,2.39,69.70,111.53,48.37],[9E9,9E9,9E9,9E9,9E9,9E9]],speeddata0,DefaultBlend,tool0;
  MoveAbsJ [[-28.31,33.79,2.21,70.69,111.80,49.13],[9E9,9E9,9E9,9E9,9E9,9E9]],speeddata0,DefaultBlend,tool0;
  MoveAbsJ [[-28.15,33.92,2.04,71.69,112.07,49.89],[9E9,9E9,9E9,9E9,9E9,9E9]],speeddata0,DefaultBlend,tool0;
  MoveAbsJ [[-28.00,34.04,1.86,72.68,112.34,50.65],[9E9,9E9,9E9,9E9,9E9,9E9]],speeddata0,FinePoint,tool0;
  TPWrite "Action 46 LinearMovement.";
  MoveAbsJ [[-28.00,34.04,1.86,72.68,112.34,50.65],[9E9,9E9,9E9,9E9,9E9,9E9]],speeddata0,DefaultBlend,tool0;
  MoveAbsJ [[-28.00,34.11,1.76,72.70,112.36,50.69],[9E9,9E9,9E9,9E9,9E9,9E9]],speeddata0,DefaultBlend,tool0;
  MoveAbsJ [[-27.97,34.67,2.02,72.40,112.10,49.85],[9E9,9E9,9E9,9E9,9E9,9E9]],speeddata0,DefaultBlend,tool0;
  MoveAbsJ [[-27.94,35.22,2.29,72.10,111.82,49.01],[9E9,9E9,9E9,9E9,9E9,9E9]],speeddata0,DefaultBlend,tool0;
  MoveAbsJ [[-27.91,35.78,2.55,71.81,111.54,48.18],[9E9,9E9,9E9,9E9,9E9,9E9]],speeddata0,DefaultBlend,tool0;
  MoveAbsJ [[-27.88,36.37,2.79,71.53,111.26,47.35],[9E9,9E9,9E9,9E9,9E9,9E9]],speeddata0,DefaultBlend,tool0;
  MoveAbsJ [[-27.85,36.96,3.00,71.25,110.98,46.53],[9E9,9E9,9E9,9E9,9E9,9E9]],speeddata0,DefaultBlend,tool0;
  MoveAbsJ [[-27.82,37.58,3.19,70.98,110.70,45.73],[9E9,9E9,9E9,9E9,9E9,9E9]],speeddata0,DefaultBlend,tool0;
  MoveAbsJ [[-27.79,38.21,3.36,70.72,110.42,44.93],[9E9,9E9,9E9,9E9,9E9,9E9]],speeddata0,DefaultBlend,tool0;
  MoveAbsJ [[-27.76,38.85,3.51,70.47,110.13,44.14],[9E9,9E9,9E9,9E9,9E9,9E9]],speeddata0,DefaultBlend,tool0;
  MoveAbsJ [[-27.73,39.51,3.64,70.23,109.85,43.37],[9E9,9E9,9E9,9E9,9E9,9E9]],speeddata0,DefaultBlend,tool0;
  MoveAbsJ [[-27.70,40.18,3.74,69.99,109.56,42.60],[9E9,9E9,9E9,9E9,9E9,9E9]],speeddata0,DefaultBlend,tool0;
  MoveAbsJ [[-27.67,40.86,3.83,69.76,109.28,41.84],[9E9,9E9,9E9,9E9,9E9,9E9]],speeddata0,DefaultBlend,tool0;
  MoveAbsJ [[-27.64,41.56,3.90,69.53,108.99,41.09],[9E9,9E9,9E9,9E9,9E9,9E9]],speeddata0,DefaultBlend,tool0;
  MoveAbsJ [[-27.61,42.27,3.94,69.31,108.71,40.35],[9E9,9E9,9E9,9E9,9E9,9E9]],speeddata0,DefaultBlend,tool0;
  MoveAbsJ [[-27.58,43.00,3.96,69.10,108.42,39.62],[9E9,9E9,9E9,9E9,9E9,9E9]],speeddata0,DefaultBlend,tool0;
  MoveAbsJ [[-27.55,43.74,3.96,68.90,108.14,38.90],[9E9,9E9,9E9,9E9,9E9,9E9]],speeddata0,DefaultBlend,tool0;
  MoveAbsJ [[-27.53,44.49,3.94,68.70,107.86,38.19],[9E9,9E9,9E9,9E9,9E9,9E9]],speeddata0,DefaultBlend,tool0;
  MoveAbsJ [[-27.50,45.26,3.89,68.51,107.58,37.49],[9E9,9E9,9E9,9E9,9E9,9E9]],speeddata0,DefaultBlend,tool0;
  MoveAbsJ [[-27.47,46.04,3.82,68.33,107.30,36.80],[9E9,9E9,9E9,9E9,9E9,9E9]],speeddata0,FinePoint,tool0;
  TPWrite "Action 47 OpenGripper.";
  TPWrite "Press Play to Continue";
  Stop;
  TPWrite "Action 48 LinearMovement.";
  MoveAbsJ [[-27.47,46.04,3.82,68.33,107.30,36.80],[9E9,9E9,9E9,9E9,9E9,9E9]],speeddata0,DefaultBlend,tool0;
  MoveAbsJ [[-28.14,46.46,3.07,67.86,107.82,36.95],[9E9,9E9,9E9,9E9,9E9,9E9]],speeddata0,DefaultBlend,tool0;
  MoveAbsJ [[-28.81,46.92,2.25,67.40,108.37,37.13],[9E9,9E9,9E9,9E9,9E9,9E9]],speeddata0,DefaultBlend,tool0;
  MoveAbsJ [[-29.48,47.40,1.40,66.96,108.91,37.32],[9E9,9E9,9E9,9E9,9E9,9E9]],speeddata0,DefaultBlend,tool0;
  MoveAbsJ [[-30.13,47.89,0.52,66.54,109.46,37.51],[9E9,9E9,9E9,9E9,9E9,9E9]],speeddata0,DefaultBlend,tool0;
  MoveAbsJ [[-30.78,48.39,-0.38,66.12,110.01,37.71],[9E9,9E9,9E9,9E9,9E9,9E9]],speeddata0,DefaultBlend,tool0;
  MoveAbsJ [[-31.42,48.91,-1.30,65.72,110.57,37.92],[9E9,9E9,9E9,9E9,9E9,9E9]],speeddata0,DefaultBlend,tool0;
  MoveAbsJ [[-32.05,49.44,-2.26,65.34,111.13,38.14],[9E9,9E9,9E9,9E9,9E9,9E9]],speeddata0,DefaultBlend,tool0;
  MoveAbsJ [[-32.67,49.99,-3.23,64.97,111.70,38.37],[9E9,9E9,9E9,9E9,9E9,9E9]],speeddata0,FinePoint,tool0;
  TPWrite "Action 49 FreeMovement.";
  MoveAbsJ [[-32.67,49.99,-3.23,64.97,111.70,38.37],[9E9,9E9,9E9,9E9,9E9,9E9]],speeddata0,DefaultBlend,tool0;
  MoveAbsJ [[-32.80,49.85,-3.00,64.81,110.71,38.57],[9E9,9E9,9E9,9E9,9E9,9E9]],speeddata0,DefaultBlend,tool0;
  MoveAbsJ [[-32.92,49.71,-2.76,64.66,109.72,38.78],[9E9,9E9,9E9,9E9,9E9,9E9]],speeddata0,DefaultBlend,tool0;
  MoveAbsJ [[-33.05,49.57,-2.52,64.50,108.73,38.98],[9E9,9E9,9E9,9E9,9E9,9E9]],speeddata0,DefaultBlend,tool0;
  MoveAbsJ [[-33.18,49.43,-2.28,64.35,107.74,39.18],[9E9,9E9,9E9,9E9,9E9,9E9]],speeddata0,DefaultBlend,tool0;
  MoveAbsJ [[-33.30,49.29,-2.04,64.19,106.75,39.38],[9E9,9E9,9E9,9E9,9E9,9E9]],speeddata0,DefaultBlend,tool0;
  MoveAbsJ [[-33.43,49.15,-1.80,64.04,105.75,39.59],[9E9,9E9,9E9,9E9,9E9,9E9]],speeddata0,DefaultBlend,tool0;
  MoveAbsJ [[-33.56,49.02,-1.56,63.89,104.76,39.79],[9E9,9E9,9E9,9E9,9E9,9E9]],speeddata0,DefaultBlend,tool0;
  MoveAbsJ [[-33.68,48.88,-1.32,63.73,103.77,39.99],[9E9,9E9,9E9,9E9,9E9,9E9]],speeddata0,DefaultBlend,tool0;
  MoveAbsJ [[-33.81,48.74,-1.08,63.58,102.78,40.19],[9E9,9E9,9E9,9E9,9E9,9E9]],speeddata0,DefaultBlend,tool0;
  MoveAbsJ [[-33.94,48.60,-0.84,63.42,101.79,40.40],[9E9,9E9,9E9,9E9,9E9,9E9]],speeddata0,DefaultBlend,tool0;
  MoveAbsJ [[-34.06,48.46,-0.60,63.27,100.80,40.60],[9E9,9E9,9E9,9E9,9E9,9E9]],speeddata0,DefaultBlend,tool0;
  MoveAbsJ [[-34.19,48.32,-0.36,63.12,99.81,40.80],[9E9,9E9,9E9,9E9,9E9,9E9]],speeddata0,DefaultBlend,tool0;
  MoveAbsJ [[-34.32,48.18,-0.12,62.96,98.82,41.01],[9E9,9E9,9E9,9E9,9E9,9E9]],speeddata0,DefaultBlend,tool0;
  MoveAbsJ [[-34.44,48.04,0.12,62.81,97.83,41.21],[9E9,9E9,9E9,9E9,9E9,9E9]],speeddata0,DefaultBlend,tool0;
  MoveAbsJ [[-34.57,47.91,0.36,62.65,96.83,41.41],[9E9,9E9,9E9,9E9,9E9,9E9]],speeddata0,DefaultBlend,tool0;
  MoveAbsJ [[-34.70,47.77,0.60,62.50,95.84,41.61],[9E9,9E9,9E9,9E9,9E9,9E9]],speeddata0,DefaultBlend,tool0;
  MoveAbsJ [[-34.82,47.63,0.83,62.35,94.85,41.82],[9E9,9E9,9E9,9E9,9E9,9E9]],speeddata0,DefaultBlend,tool0;
  MoveAbsJ [[-34.95,47.49,1.07,62.19,93.86,42.02],[9E9,9E9,9E9,9E9,9E9,9E9]],speeddata0,DefaultBlend,tool0;
  MoveAbsJ [[-35.08,47.35,1.31,62.04,92.87,42.22],[9E9,9E9,9E9,9E9,9E9,9E9]],speeddata0,DefaultBlend,tool0;
  MoveAbsJ [[-35.20,47.21,1.55,61.88,91.88,42.42],[9E9,9E9,9E9,9E9,9E9,9E9]],speeddata0,DefaultBlend,tool0;
  MoveAbsJ [[-35.33,47.07,1.79,61.73,90.89,42.63],[9E9,9E9,9E9,9E9,9E9,9E9]],speeddata0,DefaultBlend,tool0;
  MoveAbsJ [[-35.46,46.94,2.03,61.57,89.90,42.83],[9E9,9E9,9E9,9E9,9E9,9E9]],speeddata0,DefaultBlend,tool0;
  MoveAbsJ [[-35.59,46.80,2.27,61.42,88.91,43.03],[9E9,9E9,9E9,9E9,9E9,9E9]],speeddata0,DefaultBlend,tool0;
  MoveAbsJ [[-35.71,46.66,2.51,61.27,87.91,43.23],[9E9,9E9,9E9,9E9,9E9,9E9]],speeddata0,DefaultBlend,tool0;
  MoveAbsJ [[-35.84,46.52,2.75,61.11,86.92,43.44],[9E9,9E9,9E9,9E9,9E9,9E9]],speeddata0,DefaultBlend,tool0;
  MoveAbsJ [[-35.97,46.38,2.99,60.96,85.93,43.64],[9E9,9E9,9E9,9E9,9E9,9E9]],speeddata0,DefaultBlend,tool0;
  MoveAbsJ [[-36.09,46.24,3.23,60.80,84.94,43.84],[9E9,9E9,9E9,9E9,9E9,9E9]],speeddata0,DefaultBlend,tool0;
  MoveAbsJ [[-36.22,46.10,3.47,60.65,83.95,44.04],[9E9,9E9,9E9,9E9,9E9,9E9]],speeddata0,DefaultBlend,tool0;
  MoveAbsJ [[-36.35,45.96,3.71,60.50,82.96,44.25],[9E9,9E9,9E9,9E9,9E9,9E9]],speeddata0,DefaultBlend,tool0;
  MoveAbsJ [[-36.47,45.83,3.95,60.34,81.97,44.45],[9E9,9E9,9E9,9E9,9E9,9E9]],speeddata0,DefaultBlend,tool0;
  MoveAbsJ [[-36.60,45.69,4.19,60.19,80.98,44.65],[9E9,9E9,9E9,9E9,9E9,9E9]],speeddata0,DefaultBlend,tool0;
  MoveAbsJ [[-36.73,45.55,4.43,60.03,79.99,44.85],[9E9,9E9,9E9,9E9,9E9,9E9]],speeddata0,DefaultBlend,tool0;
  MoveAbsJ [[-36.85,45.41,4.67,59.88,79.00,45.06],[9E9,9E9,9E9,9E9,9E9,9E9]],speeddata0,DefaultBlend,tool0;
  MoveAbsJ [[-36.98,45.27,4.90,59.73,78.00,45.26],[9E9,9E9,9E9,9E9,9E9,9E9]],speeddata0,DefaultBlend,tool0;
  MoveAbsJ [[-37.11,45.13,5.14,59.57,77.01,45.46],[9E9,9E9,9E9,9E9,9E9,9E9]],speeddata0,DefaultBlend,tool0;
  MoveAbsJ [[-37.23,44.99,5.38,59.42,76.02,45.67],[9E9,9E9,9E9,9E9,9E9,9E9]],speeddata0,DefaultBlend,tool0;
  MoveAbsJ [[-37.36,44.86,5.62,59.26,75.03,45.87],[9E9,9E9,9E9,9E9,9E9,9E9]],speeddata0,DefaultBlend,tool0;
  MoveAbsJ [[-37.49,44.72,5.86,59.11,74.04,46.07],[9E9,9E9,9E9,9E9,9E9,9E9]],speeddata0,DefaultBlend,tool0;
  MoveAbsJ [[-37.61,44.58,6.10,58.96,73.05,46.27],[9E9,9E9,9E9,9E9,9E9,9E9]],speeddata0,DefaultBlend,tool0;
  MoveAbsJ [[-37.74,44.44,6.34,58.80,72.06,46.48],[9E9,9E9,9E9,9E9,9E9,9E9]],speeddata0,DefaultBlend,tool0;
  MoveAbsJ [[-37.87,44.30,6.58,58.65,71.07,46.68],[9E9,9E9,9E9,9E9,9E9,9E9]],speeddata0,DefaultBlend,tool0;
  MoveAbsJ [[-37.99,44.16,6.82,58.49,70.08,46.88],[9E9,9E9,9E9,9E9,9E9,9E9]],speeddata0,DefaultBlend,tool0;
  MoveAbsJ [[-38.12,44.02,7.06,58.34,69.08,47.08],[9E9,9E9,9E9,9E9,9E9,9E9]],speeddata0,DefaultBlend,tool0;
  MoveAbsJ [[-38.25,43.88,7.30,58.18,68.09,47.29],[9E9,9E9,9E9,9E9,9E9,9E9]],speeddata0,DefaultBlend,tool0;
  MoveAbsJ [[-38.37,43.75,7.54,58.03,67.10,47.49],[9E9,9E9,9E9,9E9,9E9,9E9]],speeddata0,DefaultBlend,tool0;
  MoveAbsJ [[-38.50,43.61,7.78,57.88,66.11,47.69],[9E9,9E9,9E9,9E9,9E9,9E9]],speeddata0,DefaultBlend,tool0;
  MoveAbsJ [[-38.63,43.47,8.02,57.72,65.12,47.89],[9E9,9E9,9E9,9E9,9E9,9E9]],speeddata0,DefaultBlend,tool0;
  MoveAbsJ [[-38.75,43.33,8.26,57.57,64.13,48.10],[9E9,9E9,9E9,9E9,9E9,9E9]],speeddata0,DefaultBlend,tool0;
  MoveAbsJ [[-38.88,43.19,8.50,57.41,63.14,48.30],[9E9,9E9,9E9,9E9,9E9,9E9]],speeddata0,DefaultBlend,tool0;
  MoveAbsJ [[-39.01,43.05,8.73,57.26,62.15,48.50],[9E9,9E9,9E9,9E9,9E9,9E9]],speeddata0,DefaultBlend,tool0;
  MoveAbsJ [[-39.13,42.91,8.97,57.11,61.16,48.70],[9E9,9E9,9E9,9E9,9E9,9E9]],speeddata0,DefaultBlend,tool0;
  MoveAbsJ [[-39.26,42.77,9.21,56.95,60.16,48.91],[9E9,9E9,9E9,9E9,9E9,9E9]],speeddata0,DefaultBlend,tool0;
  MoveAbsJ [[-39.39,42.64,9.45,56.80,59.17,49.11],[9E9,9E9,9E9,9E9,9E9,9E9]],speeddata0,DefaultBlend,tool0;
  MoveAbsJ [[-39.51,42.50,9.69,56.64,58.18,49.31],[9E9,9E9,9E9,9E9,9E9,9E9]],speeddata0,DefaultBlend,tool0;
  MoveAbsJ [[-39.64,42.36,9.93,56.49,57.19,49.51],[9E9,9E9,9E9,9E9,9E9,9E9]],speeddata0,DefaultBlend,tool0;
  MoveAbsJ [[-39.77,42.22,10.17,56.34,56.20,49.72],[9E9,9E9,9E9,9E9,9E9,9E9]],speeddata0,DefaultBlend,tool0;
  MoveAbsJ [[-39.90,42.08,10.41,56.18,55.21,49.92],[9E9,9E9,9E9,9E9,9E9,9E9]],speeddata0,DefaultBlend,tool0;
  MoveAbsJ [[-40.02,41.94,10.65,56.03,54.22,50.12],[9E9,9E9,9E9,9E9,9E9,9E9]],speeddata0,DefaultBlend,tool0;
  MoveAbsJ [[-40.15,41.80,10.89,55.87,53.23,50.32],[9E9,9E9,9E9,9E9,9E9,9E9]],speeddata0,DefaultBlend,tool0;
  MoveAbsJ [[-40.28,41.67,11.13,55.72,52.24,50.53],[9E9,9E9,9E9,9E9,9E9,9E9]],speeddata0,DefaultBlend,tool0;
  MoveAbsJ [[-40.40,41.53,11.37,55.56,51.24,50.73],[9E9,9E9,9E9,9E9,9E9,9E9]],speeddata0,DefaultBlend,tool0;
  MoveAbsJ [[-40.53,41.39,11.61,55.41,50.25,50.93],[9E9,9E9,9E9,9E9,9E9,9E9]],speeddata0,DefaultBlend,tool0;
  MoveAbsJ [[-40.66,41.25,11.85,55.26,49.26,51.14],[9E9,9E9,9E9,9E9,9E9,9E9]],speeddata0,DefaultBlend,tool0;
  MoveAbsJ [[-40.78,41.11,12.09,55.10,48.27,51.34],[9E9,9E9,9E9,9E9,9E9,9E9]],speeddata0,DefaultBlend,tool0;
  MoveAbsJ [[-40.91,40.97,12.33,54.95,47.28,51.54],[9E9,9E9,9E9,9E9,9E9,9E9]],speeddata0,DefaultBlend,tool0;
  MoveAbsJ [[-41.04,40.83,12.57,54.79,46.29,51.74],[9E9,9E9,9E9,9E9,9E9,9E9]],speeddata0,DefaultBlend,tool0;
  MoveAbsJ [[-41.16,40.69,12.80,54.64,45.30,51.95],[9E9,9E9,9E9,9E9,9E9,9E9]],speeddata0,DefaultBlend,tool0;
  MoveAbsJ [[-41.29,40.56,13.04,54.49,44.31,52.15],[9E9,9E9,9E9,9E9,9E9,9E9]],speeddata0,DefaultBlend,tool0;
  MoveAbsJ [[-41.42,40.42,13.28,54.33,43.32,52.35],[9E9,9E9,9E9,9E9,9E9,9E9]],speeddata0,DefaultBlend,tool0;
  MoveAbsJ [[-41.54,40.28,13.52,54.18,42.33,52.55],[9E9,9E9,9E9,9E9,9E9,9E9]],speeddata0,DefaultBlend,tool0;
  MoveAbsJ [[-41.67,40.14,13.76,54.02,41.33,52.76],[9E9,9E9,9E9,9E9,9E9,9E9]],speeddata0,DefaultBlend,tool0;
  MoveAbsJ [[-41.80,40.00,14.00,53.87,40.34,52.96],[9E9,9E9,9E9,9E9,9E9,9E9]],speeddata0,DefaultBlend,tool0;
  MoveAbsJ [[-41.92,39.86,14.24,53.72,39.35,53.16],[9E9,9E9,9E9,9E9,9E9,9E9]],speeddata0,DefaultBlend,tool0;
  MoveAbsJ [[-42.05,39.72,14.48,53.56,38.36,53.36],[9E9,9E9,9E9,9E9,9E9,9E9]],speeddata0,DefaultBlend,tool0;
  MoveAbsJ [[-42.18,39.59,14.72,53.41,37.37,53.57],[9E9,9E9,9E9,9E9,9E9,9E9]],speeddata0,DefaultBlend,tool0;
  MoveAbsJ [[-42.30,39.45,14.96,53.25,36.38,53.77],[9E9,9E9,9E9,9E9,9E9,9E9]],speeddata0,DefaultBlend,tool0;
  MoveAbsJ [[-42.43,39.31,15.20,53.10,35.39,53.97],[9E9,9E9,9E9,9E9,9E9,9E9]],speeddata0,DefaultBlend,tool0;
  MoveAbsJ [[-42.56,39.17,15.44,52.94,34.40,54.17],[9E9,9E9,9E9,9E9,9E9,9E9]],speeddata0,DefaultBlend,tool0;
  MoveAbsJ [[-42.68,39.03,15.68,52.79,33.41,54.38],[9E9,9E9,9E9,9E9,9E9,9E9]],speeddata0,DefaultBlend,tool0;
  MoveAbsJ [[-42.81,38.89,15.92,52.64,32.41,54.58],[9E9,9E9,9E9,9E9,9E9,9E9]],speeddata0,DefaultBlend,tool0;
  MoveAbsJ [[-42.94,38.75,16.16,52.48,31.42,54.78],[9E9,9E9,9E9,9E9,9E9,9E9]],speeddata0,DefaultBlend,tool0;
  MoveAbsJ [[-43.06,38.61,16.40,52.33,30.43,54.98],[9E9,9E9,9E9,9E9,9E9,9E9]],speeddata0,DefaultBlend,tool0;
  MoveAbsJ [[-43.19,38.48,16.63,52.17,29.44,55.19],[9E9,9E9,9E9,9E9,9E9,9E9]],speeddata0,DefaultBlend,tool0;
  MoveAbsJ [[-43.32,38.34,16.87,52.02,28.45,55.39],[9E9,9E9,9E9,9E9,9E9,9E9]],speeddata0,DefaultBlend,tool0;
  MoveAbsJ [[-43.44,38.20,17.11,51.87,27.46,55.59],[9E9,9E9,9E9,9E9,9E9,9E9]],speeddata0,DefaultBlend,tool0;
  MoveAbsJ [[-43.57,38.06,17.35,51.71,26.47,55.80],[9E9,9E9,9E9,9E9,9E9,9E9]],speeddata0,DefaultBlend,tool0;
  MoveAbsJ [[-43.70,37.92,17.59,51.56,25.48,56.00],[9E9,9E9,9E9,9E9,9E9,9E9]],speeddata0,DefaultBlend,tool0;
  MoveAbsJ [[-43.82,37.78,17.83,51.40,24.49,56.20],[9E9,9E9,9E9,9E9,9E9,9E9]],speeddata0,DefaultBlend,tool0;
  MoveAbsJ [[-43.95,37.64,18.07,51.25,23.49,56.40],[9E9,9E9,9E9,9E9,9E9,9E9]],speeddata0,DefaultBlend,tool0;
  MoveAbsJ [[-44.08,37.51,18.31,51.10,22.50,56.61],[9E9,9E9,9E9,9E9,9E9,9E9]],speeddata0,DefaultBlend,tool0;
  MoveAbsJ [[-44.20,37.37,18.55,50.94,21.51,56.81],[9E9,9E9,9E9,9E9,9E9,9E9]],speeddata0,DefaultBlend,tool0;
  MoveAbsJ [[-44.33,37.23,18.79,50.79,20.52,57.01],[9E9,9E9,9E9,9E9,9E9,9E9]],speeddata0,DefaultBlend,tool0;
  MoveAbsJ [[-44.46,37.09,19.03,50.63,19.53,57.21],[9E9,9E9,9E9,9E9,9E9,9E9]],speeddata0,DefaultBlend,tool0;
  MoveAbsJ [[-44.59,36.95,19.27,50.48,18.54,57.42],[9E9,9E9,9E9,9E9,9E9,9E9]],speeddata0,DefaultBlend,tool0;
  MoveAbsJ [[-44.71,36.81,19.51,50.33,17.55,57.62],[9E9,9E9,9E9,9E9,9E9,9E9]],speeddata0,DefaultBlend,tool0;
  MoveAbsJ [[-44.84,36.67,19.75,50.17,16.56,57.82],[9E9,9E9,9E9,9E9,9E9,9E9]],speeddata0,DefaultBlend,tool0;
  MoveAbsJ [[-44.97,36.53,19.99,50.02,15.57,58.02],[9E9,9E9,9E9,9E9,9E9,9E9]],speeddata0,DefaultBlend,tool0;
  MoveAbsJ [[-45.09,36.40,20.23,49.86,14.57,58.23],[9E9,9E9,9E9,9E9,9E9,9E9]],speeddata0,DefaultBlend,tool0;
  MoveAbsJ [[-45.22,36.26,20.47,49.71,13.58,58.43],[9E9,9E9,9E9,9E9,9E9,9E9]],speeddata0,DefaultBlend,tool0;
  MoveAbsJ [[-45.35,36.12,20.70,49.55,12.59,58.63],[9E9,9E9,9E9,9E9,9E9,9E9]],speeddata0,DefaultBlend,tool0;
  MoveAbsJ [[-45.47,35.98,20.94,49.40,11.60,58.83],[9E9,9E9,9E9,9E9,9E9,9E9]],speeddata0,DefaultBlend,tool0;
  MoveAbsJ [[-45.60,35.84,21.18,49.25,10.61,59.04],[9E9,9E9,9E9,9E9,9E9,9E9]],speeddata0,DefaultBlend,tool0;
  MoveAbsJ [[-45.73,35.70,21.42,49.09,9.62,59.24],[9E9,9E9,9E9,9E9,9E9,9E9]],speeddata0,DefaultBlend,tool0;
  MoveAbsJ [[-45.85,35.56,21.66,48.94,8.63,59.44],[9E9,9E9,9E9,9E9,9E9,9E9]],speeddata0,DefaultBlend,tool0;
  MoveAbsJ [[-45.98,35.42,21.90,48.78,7.64,59.64],[9E9,9E9,9E9,9E9,9E9,9E9]],speeddata0,DefaultBlend,tool0;
  MoveAbsJ [[-46.11,35.29,22.14,48.63,6.65,59.85],[9E9,9E9,9E9,9E9,9E9,9E9]],speeddata0,DefaultBlend,tool0;
  MoveAbsJ [[-46.23,35.15,22.38,48.48,5.66,60.05],[9E9,9E9,9E9,9E9,9E9,9E9]],speeddata0,DefaultBlend,tool0;
  MoveAbsJ [[-46.36,35.01,22.62,48.32,4.66,60.25],[9E9,9E9,9E9,9E9,9E9,9E9]],speeddata0,DefaultBlend,tool0;
  MoveAbsJ [[-46.49,34.87,22.86,48.17,3.67,60.45],[9E9,9E9,9E9,9E9,9E9,9E9]],speeddata0,DefaultBlend,tool0;
  MoveAbsJ [[-46.61,34.73,23.10,48.01,2.68,60.66],[9E9,9E9,9E9,9E9,9E9,9E9]],speeddata0,DefaultBlend,tool0;
  MoveAbsJ [[-46.74,34.59,23.34,47.86,1.69,60.86],[9E9,9E9,9E9,9E9,9E9,9E9]],speeddata0,DefaultBlend,tool0;
  MoveAbsJ [[-46.87,34.45,23.58,47.71,0.70,61.06],[9E9,9E9,9E9,9E9,9E9,9E9]],speeddata0,DefaultBlend,tool0;
  MoveAbsJ [[-46.99,34.32,23.82,47.55,-0.29,61.27],[9E9,9E9,9E9,9E9,9E9,9E9]],speeddata0,DefaultBlend,tool0;
  MoveAbsJ [[-47.12,34.18,24.06,47.40,-1.28,61.47],[9E9,9E9,9E9,9E9,9E9,9E9]],speeddata0,DefaultBlend,tool0;
  MoveAbsJ [[-47.25,34.04,24.30,47.24,-2.27,61.67],[9E9,9E9,9E9,9E9,9E9,9E9]],speeddata0,DefaultBlend,tool0;
  MoveAbsJ [[-47.37,33.90,24.53,47.09,-3.26,61.87],[9E9,9E9,9E9,9E9,9E9,9E9]],speeddata0,DefaultBlend,tool0;
  MoveAbsJ [[-47.50,33.76,24.77,46.93,-4.26,62.08],[9E9,9E9,9E9,9E9,9E9,9E9]],speeddata0,DefaultBlend,tool0;
  MoveAbsJ [[-47.63,33.62,25.01,46.78,-5.25,62.28],[9E9,9E9,9E9,9E9,9E9,9E9]],speeddata0,DefaultBlend,tool0;
  MoveAbsJ [[-47.75,33.48,25.25,46.63,-6.24,62.48],[9E9,9E9,9E9,9E9,9E9,9E9]],speeddata0,DefaultBlend,tool0;
  MoveAbsJ [[-47.88,33.34,25.49,46.47,-7.23,62.68],[9E9,9E9,9E9,9E9,9E9,9E9]],speeddata0,DefaultBlend,tool0;
  MoveAbsJ [[-48.01,33.21,25.73,46.32,-8.22,62.89],[9E9,9E9,9E9,9E9,9E9,9E9]],speeddata0,DefaultBlend,tool0;
  MoveAbsJ [[-48.13,33.07,25.97,46.16,-9.21,63.09],[9E9,9E9,9E9,9E9,9E9,9E9]],speeddata0,DefaultBlend,tool0;
  MoveAbsJ [[-48.26,32.93,26.21,46.01,-10.20,63.29],[9E9,9E9,9E9,9E9,9E9,9E9]],speeddata0,DefaultBlend,tool0;
  MoveAbsJ [[-48.39,32.79,26.45,45.86,-11.19,63.49],[9E9,9E9,9E9,9E9,9E9,9E9]],speeddata0,DefaultBlend,tool0;
  MoveAbsJ [[-48.51,32.65,26.69,45.70,-12.18,63.70],[9E9,9E9,9E9,9E9,9E9,9E9]],speeddata0,DefaultBlend,tool0;
  MoveAbsJ [[-48.64,32.51,26.93,45.55,-13.18,63.90],[9E9,9E9,9E9,9E9,9E9,9E9]],speeddata0,DefaultBlend,tool0;
  MoveAbsJ [[-48.77,32.37,27.17,45.39,-14.17,64.10],[9E9,9E9,9E9,9E9,9E9,9E9]],speeddata0,DefaultBlend,tool0;
  MoveAbsJ [[-48.90,32.24,27.41,45.24,-15.16,64.30],[9E9,9E9,9E9,9E9,9E9,9E9]],speeddata0,DefaultBlend,tool0;
  MoveAbsJ [[-49.02,32.10,27.65,45.09,-16.15,64.51],[9E9,9E9,9E9,9E9,9E9,9E9]],speeddata0,DefaultBlend,tool0;
  MoveAbsJ [[-49.15,31.96,27.89,44.93,-17.14,64.71],[9E9,9E9,9E9,9E9,9E9,9E9]],speeddata0,DefaultBlend,tool0;
  MoveAbsJ [[-49.28,31.82,28.13,44.78,-18.13,64.91],[9E9,9E9,9E9,9E9,9E9,9E9]],speeddata0,DefaultBlend,tool0;
  MoveAbsJ [[-49.40,31.68,28.37,44.62,-19.12,65.11],[9E9,9E9,9E9,9E9,9E9,9E9]],speeddata0,DefaultBlend,tool0;
  MoveAbsJ [[-49.53,31.54,28.60,44.47,-20.11,65.32],[9E9,9E9,9E9,9E9,9E9,9E9]],speeddata0,DefaultBlend,tool0;
  MoveAbsJ [[-49.66,31.40,28.84,44.31,-21.10,65.52],[9E9,9E9,9E9,9E9,9E9,9E9]],speeddata0,DefaultBlend,tool0;
  MoveAbsJ [[-49.78,31.26,29.08,44.16,-22.10,65.72],[9E9,9E9,9E9,9E9,9E9,9E9]],speeddata0,DefaultBlend,tool0;
  MoveAbsJ [[-49.91,31.13,29.32,44.01,-23.09,65.93],[9E9,9E9,9E9,9E9,9E9,9E9]],speeddata0,DefaultBlend,tool0;
  MoveAbsJ [[-50.04,30.99,29.56,43.85,-24.08,66.13],[9E9,9E9,9E9,9E9,9E9,9E9]],speeddata0,DefaultBlend,tool0;
  MoveAbsJ [[-50.16,30.85,29.80,43.70,-25.07,66.33],[9E9,9E9,9E9,9E9,9E9,9E9]],speeddata0,DefaultBlend,tool0;
  MoveAbsJ [[-50.29,30.71,30.04,43.54,-26.06,66.53],[9E9,9E9,9E9,9E9,9E9,9E9]],speeddata0,DefaultBlend,tool0;
  MoveAbsJ [[-50.42,30.57,30.28,43.39,-27.05,66.74],[9E9,9E9,9E9,9E9,9E9,9E9]],speeddata0,DefaultBlend,tool0;
  MoveAbsJ [[-50.54,30.43,30.52,43.24,-28.04,66.94],[9E9,9E9,9E9,9E9,9E9,9E9]],speeddata0,DefaultBlend,tool0;
  MoveAbsJ [[-50.67,30.29,30.76,43.08,-29.03,67.14],[9E9,9E9,9E9,9E9,9E9,9E9]],speeddata0,DefaultBlend,tool0;
  MoveAbsJ [[-50.80,30.16,31.00,42.93,-30.02,67.34],[9E9,9E9,9E9,9E9,9E9,9E9]],speeddata0,DefaultBlend,tool0;
  MoveAbsJ [[-50.92,30.02,31.24,42.77,-31.01,67.55],[9E9,9E9,9E9,9E9,9E9,9E9]],speeddata0,DefaultBlend,tool0;
  MoveAbsJ [[-51.05,29.88,31.48,42.62,-32.01,67.75],[9E9,9E9,9E9,9E9,9E9,9E9]],speeddata0,DefaultBlend,tool0;
  MoveAbsJ [[-51.18,29.74,31.72,42.47,-33.00,67.95],[9E9,9E9,9E9,9E9,9E9,9E9]],speeddata0,DefaultBlend,tool0;
  MoveAbsJ [[-51.30,29.60,31.96,42.31,-33.99,68.15],[9E9,9E9,9E9,9E9,9E9,9E9]],speeddata0,DefaultBlend,tool0;
  MoveAbsJ [[-51.43,29.46,32.20,42.16,-34.98,68.36],[9E9,9E9,9E9,9E9,9E9,9E9]],speeddata0,DefaultBlend,tool0;
  MoveAbsJ [[-51.56,29.32,32.43,42.00,-35.97,68.56],[9E9,9E9,9E9,9E9,9E9,9E9]],speeddata0,DefaultBlend,tool0;
  MoveAbsJ [[-51.68,29.18,32.67,41.85,-36.96,68.76],[9E9,9E9,9E9,9E9,9E9,9E9]],speeddata0,DefaultBlend,tool0;
  MoveAbsJ [[-51.81,29.05,32.91,41.70,-37.95,68.96],[9E9,9E9,9E9,9E9,9E9,9E9]],speeddata0,DefaultBlend,tool0;
  MoveAbsJ [[-51.94,28.91,33.15,41.54,-38.94,69.17],[9E9,9E9,9E9,9E9,9E9,9E9]],speeddata0,DefaultBlend,tool0;
  MoveAbsJ [[-52.06,28.77,33.39,41.39,-39.93,69.37],[9E9,9E9,9E9,9E9,9E9,9E9]],speeddata0,DefaultBlend,tool0;
  MoveAbsJ [[-52.19,28.63,33.63,41.23,-40.93,69.57],[9E9,9E9,9E9,9E9,9E9,9E9]],speeddata0,DefaultBlend,tool0;
  MoveAbsJ [[-52.32,28.49,33.87,41.08,-41.92,69.77],[9E9,9E9,9E9,9E9,9E9,9E9]],speeddata0,DefaultBlend,tool0;
  MoveAbsJ [[-52.44,28.35,34.11,40.92,-42.91,69.98],[9E9,9E9,9E9,9E9,9E9,9E9]],speeddata0,DefaultBlend,tool0;
  MoveAbsJ [[-52.57,28.21,34.35,40.77,-43.90,70.18],[9E9,9E9,9E9,9E9,9E9,9E9]],speeddata0,DefaultBlend,tool0;
  MoveAbsJ [[-52.70,28.07,34.59,40.62,-44.89,70.38],[9E9,9E9,9E9,9E9,9E9,9E9]],speeddata0,DefaultBlend,tool0;
  MoveAbsJ [[-52.82,27.94,34.83,40.46,-45.88,70.58],[9E9,9E9,9E9,9E9,9E9,9E9]],speeddata0,DefaultBlend,tool0;
  MoveAbsJ [[-52.95,27.80,35.07,40.31,-46.87,70.79],[9E9,9E9,9E9,9E9,9E9,9E9]],speeddata0,DefaultBlend,tool0;
  MoveAbsJ [[-53.08,27.66,35.31,40.15,-47.86,70.99],[9E9,9E9,9E9,9E9,9E9,9E9]],speeddata0,DefaultBlend,tool0;
  MoveAbsJ [[-53.21,27.52,35.55,40.00,-48.85,71.19],[9E9,9E9,9E9,9E9,9E9,9E9]],speeddata0,DefaultBlend,tool0;
  MoveAbsJ [[-53.33,27.38,35.79,39.85,-49.85,71.40],[9E9,9E9,9E9,9E9,9E9,9E9]],speeddata0,DefaultBlend,tool0;
  MoveAbsJ [[-53.46,27.24,36.03,39.69,-50.84,71.60],[9E9,9E9,9E9,9E9,9E9,9E9]],speeddata0,DefaultBlend,tool0;
  MoveAbsJ [[-53.59,27.10,36.27,39.54,-51.83,71.80],[9E9,9E9,9E9,9E9,9E9,9E9]],speeddata0,DefaultBlend,tool0;
  MoveAbsJ [[-53.71,26.97,36.50,39.38,-52.82,72.00],[9E9,9E9,9E9,9E9,9E9,9E9]],speeddata0,DefaultBlend,tool0;
  MoveAbsJ [[-53.84,26.83,36.74,39.23,-53.81,72.21],[9E9,9E9,9E9,9E9,9E9,9E9]],speeddata0,DefaultBlend,tool0;
  MoveAbsJ [[-53.97,26.69,36.98,39.08,-54.80,72.41],[9E9,9E9,9E9,9E9,9E9,9E9]],speeddata0,DefaultBlend,tool0;
  MoveAbsJ [[-54.09,26.55,37.22,38.92,-55.79,72.61],[9E9,9E9,9E9,9E9,9E9,9E9]],speeddata0,DefaultBlend,tool0;
  MoveAbsJ [[-54.22,26.41,37.46,38.77,-56.78,72.81],[9E9,9E9,9E9,9E9,9E9,9E9]],speeddata0,DefaultBlend,tool0;
  MoveAbsJ [[-54.35,26.27,37.70,38.61,-57.77,73.02],[9E9,9E9,9E9,9E9,9E9,9E9]],speeddata0,DefaultBlend,tool0;
  MoveAbsJ [[-54.47,26.13,37.94,38.46,-58.77,73.22],[9E9,9E9,9E9,9E9,9E9,9E9]],speeddata0,DefaultBlend,tool0;
  MoveAbsJ [[-54.60,25.99,38.18,38.30,-59.76,73.42],[9E9,9E9,9E9,9E9,9E9,9E9]],speeddata0,DefaultBlend,tool0;
  MoveAbsJ [[-54.73,25.86,38.42,38.15,-60.75,73.62],[9E9,9E9,9E9,9E9,9E9,9E9]],speeddata0,DefaultBlend,tool0;
  MoveAbsJ [[-54.85,25.72,38.66,38.00,-61.74,73.83],[9E9,9E9,9E9,9E9,9E9,9E9]],speeddata0,DefaultBlend,tool0;
  MoveAbsJ [[-54.98,25.58,38.90,37.84,-62.73,74.03],[9E9,9E9,9E9,9E9,9E9,9E9]],speeddata0,DefaultBlend,tool0;
  MoveAbsJ [[-55.11,25.44,39.14,37.69,-63.72,74.23],[9E9,9E9,9E9,9E9,9E9,9E9]],speeddata0,DefaultBlend,tool0;
  MoveAbsJ [[-55.23,25.30,39.38,37.53,-64.71,74.43],[9E9,9E9,9E9,9E9,9E9,9E9]],speeddata0,DefaultBlend,tool0;
  MoveAbsJ [[-55.36,25.16,39.62,37.38,-65.70,74.64],[9E9,9E9,9E9,9E9,9E9,9E9]],speeddata0,DefaultBlend,tool0;
  MoveAbsJ [[-55.49,25.02,39.86,37.23,-66.69,74.84],[9E9,9E9,9E9,9E9,9E9,9E9]],speeddata0,DefaultBlend,tool0;
  MoveAbsJ [[-55.61,24.89,40.10,37.07,-67.68,75.04],[9E9,9E9,9E9,9E9,9E9,9E9]],speeddata0,DefaultBlend,tool0;
  MoveAbsJ [[-55.74,24.75,40.33,36.92,-68.68,75.24],[9E9,9E9,9E9,9E9,9E9,9E9]],speeddata0,DefaultBlend,tool0;
  MoveAbsJ [[-55.87,24.61,40.57,36.76,-69.67,75.45],[9E9,9E9,9E9,9E9,9E9,9E9]],speeddata0,FinePoint,tool0;
  TPWrite "Action 50 LoadWorkpiece.";
  TPWrite "Press Play to Continue";
  Stop;
  TPWrite "Action 51 CloseGripper.";
  TPWrite "Press Play to Continue";
  Stop;
  TPWrite "Action 52 FreeMovement.";
  MoveAbsJ [[-55.87,24.61,40.57,36.76,-69.67,75.45],[9E9,9E9,9E9,9E9,9E9,9E9]],speeddata0,DefaultBlend,tool0;
  MoveAbsJ [[-54.88,23.93,39.58,35.90,-69.56,75.66],[9E9,9E9,9E9,9E9,9E9,9E9]],speeddata0,DefaultBlend,tool0;
  MoveAbsJ [[-53.90,23.25,38.59,35.04,-69.45,75.88],[9E9,9E9,9E9,9E9,9E9,9E9]],speeddata0,DefaultBlend,tool0;
  MoveAbsJ [[-52.91,22.58,37.60,34.17,-69.33,76.10],[9E9,9E9,9E9,9E9,9E9,9E9]],speeddata0,DefaultBlend,tool0;
  MoveAbsJ [[-51.93,21.90,36.61,33.31,-69.22,76.32],[9E9,9E9,9E9,9E9,9E9,9E9]],speeddata0,DefaultBlend,tool0;
  MoveAbsJ [[-50.95,21.22,35.62,32.45,-69.11,76.53],[9E9,9E9,9E9,9E9,9E9,9E9]],speeddata0,DefaultBlend,tool0;
  MoveAbsJ [[-49.96,20.55,34.63,31.58,-69.00,76.75],[9E9,9E9,9E9,9E9,9E9,9E9]],speeddata0,DefaultBlend,tool0;
  MoveAbsJ [[-48.98,19.87,33.64,30.72,-68.89,76.97],[9E9,9E9,9E9,9E9,9E9,9E9]],speeddata0,DefaultBlend,tool0;
  MoveAbsJ [[-47.99,19.19,32.65,29.86,-68.78,77.19],[9E9,9E9,9E9,9E9,9E9,9E9]],speeddata0,DefaultBlend,tool0;
  MoveAbsJ [[-47.01,18.51,31.65,28.99,-68.67,77.40],[9E9,9E9,9E9,9E9,9E9,9E9]],speeddata0,DefaultBlend,tool0;
  MoveAbsJ [[-46.02,17.84,30.66,28.13,-68.56,77.62],[9E9,9E9,9E9,9E9,9E9,9E9]],speeddata0,DefaultBlend,tool0;
  MoveAbsJ [[-45.04,17.16,29.67,27.27,-68.45,77.84],[9E9,9E9,9E9,9E9,9E9,9E9]],speeddata0,DefaultBlend,tool0;
  MoveAbsJ [[-44.06,16.48,28.68,26.40,-68.34,78.06],[9E9,9E9,9E9,9E9,9E9,9E9]],speeddata0,DefaultBlend,tool0;
  MoveAbsJ [[-43.07,15.81,27.69,25.54,-68.22,78.27],[9E9,9E9,9E9,9E9,9E9,9E9]],speeddata0,DefaultBlend,tool0;
  MoveAbsJ [[-42.09,15.13,26.70,24.68,-68.11,78.49],[9E9,9E9,9E9,9E9,9E9,9E9]],speeddata0,DefaultBlend,tool0;
  MoveAbsJ [[-41.10,14.45,25.71,23.81,-68.00,78.71],[9E9,9E9,9E9,9E9,9E9,9E9]],speeddata0,DefaultBlend,tool0;
  MoveAbsJ [[-40.12,13.78,24.72,22.95,-67.89,78.93],[9E9,9E9,9E9,9E9,9E9,9E9]],speeddata0,DefaultBlend,tool0;
  MoveAbsJ [[-39.14,13.10,23.73,22.09,-67.78,79.14],[9E9,9E9,9E9,9E9,9E9,9E9]],speeddata0,DefaultBlend,tool0;
  MoveAbsJ [[-38.15,12.42,22.73,21.22,-67.67,79.36],[9E9,9E9,9E9,9E9,9E9,9E9]],speeddata0,DefaultBlend,tool0;
  MoveAbsJ [[-37.17,11.75,21.74,20.36,-67.56,79.58],[9E9,9E9,9E9,9E9,9E9,9E9]],speeddata0,DefaultBlend,tool0;
  MoveAbsJ [[-36.18,11.07,20.75,19.50,-67.45,79.79],[9E9,9E9,9E9,9E9,9E9,9E9]],speeddata0,DefaultBlend,tool0;
  MoveAbsJ [[-35.20,10.39,19.76,18.63,-67.34,80.01],[9E9,9E9,9E9,9E9,9E9,9E9]],speeddata0,DefaultBlend,tool0;
  MoveAbsJ [[-34.21,9.71,18.77,17.77,-67.23,80.23],[9E9,9E9,9E9,9E9,9E9,9E9]],speeddata0,DefaultBlend,tool0;
  MoveAbsJ [[-33.23,9.04,17.78,16.91,-67.12,80.45],[9E9,9E9,9E9,9E9,9E9,9E9]],speeddata0,DefaultBlend,tool0;
  MoveAbsJ [[-32.74,8.70,17.28,16.48,-67.06,80.56],[9E9,9E9,9E9,9E9,9E9,9E9]],speeddata0,DefaultBlend,tool0;
  MoveAbsJ [[-31.81,8.27,16.71,17.38,-66.08,80.78],[9E9,9E9,9E9,9E9,9E9,9E9]],speeddata0,DefaultBlend,tool0;
  MoveAbsJ [[-30.88,7.84,16.13,18.29,-65.11,81.01],[9E9,9E9,9E9,9E9,9E9,9E9]],speeddata0,DefaultBlend,tool0;
  MoveAbsJ [[-30.64,7.82,16.15,19.28,-64.47,81.07],[9E9,9E9,9E9,9E9,9E9,9E9]],speeddata0,DefaultBlend,tool0;
  MoveAbsJ [[-30.40,7.80,16.16,20.27,-63.83,81.14],[9E9,9E9,9E9,9E9,9E9,9E9]],speeddata0,DefaultBlend,tool0;
  MoveAbsJ [[-30.17,7.78,16.17,21.26,-63.20,81.21],[9E9,9E9,9E9,9E9,9E9,9E9]],speeddata0,DefaultBlend,tool0;
  MoveAbsJ [[-29.93,7.77,16.18,22.25,-62.56,81.27],[9E9,9E9,9E9,9E9,9E9,9E9]],speeddata0,DefaultBlend,tool0;
  MoveAbsJ [[-29.69,7.75,16.19,23.25,-61.92,81.34],[9E9,9E9,9E9,9E9,9E9,9E9]],speeddata0,DefaultBlend,tool0;
  MoveAbsJ [[-29.45,7.73,16.21,24.24,-61.29,81.41],[9E9,9E9,9E9,9E9,9E9,9E9]],speeddata0,DefaultBlend,tool0;
  MoveAbsJ [[-29.21,7.71,16.22,25.23,-60.65,81.47],[9E9,9E9,9E9,9E9,9E9,9E9]],speeddata0,DefaultBlend,tool0;
  MoveAbsJ [[-28.97,7.69,16.23,26.22,-60.01,81.54],[9E9,9E9,9E9,9E9,9E9,9E9]],speeddata0,DefaultBlend,tool0;
  MoveAbsJ [[-28.73,7.67,16.24,27.21,-59.38,81.61],[9E9,9E9,9E9,9E9,9E9,9E9]],speeddata0,DefaultBlend,tool0;
  MoveAbsJ [[-28.50,7.66,16.25,28.21,-58.74,81.67],[9E9,9E9,9E9,9E9,9E9,9E9]],speeddata0,DefaultBlend,tool0;
  MoveAbsJ [[-28.26,7.64,16.27,29.20,-58.10,81.74],[9E9,9E9,9E9,9E9,9E9,9E9]],speeddata0,DefaultBlend,tool0;
  MoveAbsJ [[-28.02,7.62,16.28,30.19,-57.47,81.80],[9E9,9E9,9E9,9E9,9E9,9E9]],speeddata0,DefaultBlend,tool0;
  MoveAbsJ [[-27.78,7.60,16.29,31.18,-56.83,81.87],[9E9,9E9,9E9,9E9,9E9,9E9]],speeddata0,DefaultBlend,tool0;
  MoveAbsJ [[-27.54,7.58,16.30,32.18,-56.20,81.94],[9E9,9E9,9E9,9E9,9E9,9E9]],speeddata0,DefaultBlend,tool0;
  MoveAbsJ [[-27.30,7.56,16.31,33.17,-55.56,82.00],[9E9,9E9,9E9,9E9,9E9,9E9]],speeddata0,DefaultBlend,tool0;
  MoveAbsJ [[-27.07,7.55,16.33,34.16,-54.92,82.07],[9E9,9E9,9E9,9E9,9E9,9E9]],speeddata0,DefaultBlend,tool0;
  MoveAbsJ [[-26.83,7.53,16.34,35.15,-54.29,82.14],[9E9,9E9,9E9,9E9,9E9,9E9]],speeddata0,DefaultBlend,tool0;
  MoveAbsJ [[-26.59,7.51,16.35,36.14,-53.65,82.20],[9E9,9E9,9E9,9E9,9E9,9E9]],speeddata0,DefaultBlend,tool0;
  MoveAbsJ [[-26.35,7.49,16.36,37.14,-53.01,82.27],[9E9,9E9,9E9,9E9,9E9,9E9]],speeddata0,DefaultBlend,tool0;
  MoveAbsJ [[-26.11,7.47,16.37,38.13,-52.38,82.34],[9E9,9E9,9E9,9E9,9E9,9E9]],speeddata0,DefaultBlend,tool0;
  MoveAbsJ [[-25.87,7.46,16.39,39.12,-51.74,82.40],[9E9,9E9,9E9,9E9,9E9,9E9]],speeddata0,DefaultBlend,tool0;
  MoveAbsJ [[-25.64,7.44,16.40,40.11,-51.10,82.47],[9E9,9E9,9E9,9E9,9E9,9E9]],speeddata0,DefaultBlend,tool0;
  MoveAbsJ [[-25.40,7.42,16.41,41.11,-50.47,82.54],[9E9,9E9,9E9,9E9,9E9,9E9]],speeddata0,DefaultBlend,tool0;
  MoveAbsJ [[-25.16,7.40,16.42,42.10,-49.83,82.60],[9E9,9E9,9E9,9E9,9E9,9E9]],speeddata0,DefaultBlend,tool0;
  MoveAbsJ [[-24.92,7.38,16.43,43.09,-49.19,82.67],[9E9,9E9,9E9,9E9,9E9,9E9]],speeddata0,DefaultBlend,tool0;
  MoveAbsJ [[-24.68,7.36,16.45,44.08,-48.56,82.74],[9E9,9E9,9E9,9E9,9E9,9E9]],speeddata0,DefaultBlend,tool0;
  MoveAbsJ [[-24.44,7.35,16.46,45.07,-47.92,82.80],[9E9,9E9,9E9,9E9,9E9,9E9]],speeddata0,DefaultBlend,tool0;
  MoveAbsJ [[-24.20,7.33,16.47,46.07,-47.28,82.87],[9E9,9E9,9E9,9E9,9E9,9E9]],speeddata0,DefaultBlend,tool0;
  MoveAbsJ [[-23.97,7.31,16.48,47.06,-46.65,82.94],[9E9,9E9,9E9,9E9,9E9,9E9]],speeddata0,DefaultBlend,tool0;
  MoveAbsJ [[-23.73,7.29,16.49,48.05,-46.01,83.00],[9E9,9E9,9E9,9E9,9E9,9E9]],speeddata0,DefaultBlend,tool0;
  MoveAbsJ [[-23.49,7.27,16.51,49.04,-45.38,83.07],[9E9,9E9,9E9,9E9,9E9,9E9]],speeddata0,DefaultBlend,tool0;
  MoveAbsJ [[-23.25,7.25,16.52,50.04,-44.74,83.14],[9E9,9E9,9E9,9E9,9E9,9E9]],speeddata0,DefaultBlend,tool0;
  MoveAbsJ [[-23.01,7.24,16.53,51.03,-44.10,83.20],[9E9,9E9,9E9,9E9,9E9,9E9]],speeddata0,DefaultBlend,tool0;
  MoveAbsJ [[-22.77,7.22,16.54,52.02,-43.47,83.27],[9E9,9E9,9E9,9E9,9E9,9E9]],speeddata0,DefaultBlend,tool0;
  MoveAbsJ [[-22.54,7.20,16.55,53.01,-42.83,83.34],[9E9,9E9,9E9,9E9,9E9,9E9]],speeddata0,DefaultBlend,tool0;
  MoveAbsJ [[-22.30,7.18,16.57,54.00,-42.19,83.40],[9E9,9E9,9E9,9E9,9E9,9E9]],speeddata0,DefaultBlend,tool0;
  MoveAbsJ [[-22.06,7.16,16.58,55.00,-41.56,83.47],[9E9,9E9,9E9,9E9,9E9,9E9]],speeddata0,DefaultBlend,tool0;
  MoveAbsJ [[-21.82,7.14,16.59,55.99,-40.92,83.54],[9E9,9E9,9E9,9E9,9E9,9E9]],speeddata0,DefaultBlend,tool0;
  MoveAbsJ [[-21.58,7.13,16.60,56.98,-40.28,83.60],[9E9,9E9,9E9,9E9,9E9,9E9]],speeddata0,DefaultBlend,tool0;
  MoveAbsJ [[-21.34,7.11,16.61,57.97,-39.65,83.67],[9E9,9E9,9E9,9E9,9E9,9E9]],speeddata0,DefaultBlend,tool0;
  MoveAbsJ [[-21.10,7.09,16.63,58.97,-39.01,83.74],[9E9,9E9,9E9,9E9,9E9,9E9]],speeddata0,DefaultBlend,tool0;
  MoveAbsJ [[-20.87,7.07,16.64,59.96,-38.37,83.80],[9E9,9E9,9E9,9E9,9E9,9E9]],speeddata0,DefaultBlend,tool0;
  MoveAbsJ [[-20.63,7.05,16.65,60.95,-37.74,83.87],[9E9,9E9,9E9,9E9,9E9,9E9]],speeddata0,DefaultBlend,tool0;
  MoveAbsJ [[-20.39,7.04,16.66,61.94,-37.10,83.94],[9E9,9E9,9E9,9E9,9E9,9E9]],speeddata0,DefaultBlend,tool0;
  MoveAbsJ [[-20.15,7.02,16.67,62.93,-36.47,84.00],[9E9,9E9,9E9,9E9,9E9,9E9]],speeddata0,DefaultBlend,tool0;
  MoveAbsJ [[-19.91,7.00,16.69,63.93,-35.83,84.07],[9E9,9E9,9E9,9E9,9E9,9E9]],speeddata0,DefaultBlend,tool0;
  MoveAbsJ [[-19.67,6.98,16.70,64.92,-35.19,84.14],[9E9,9E9,9E9,9E9,9E9,9E9]],speeddata0,DefaultBlend,tool0;
  MoveAbsJ [[-19.44,6.96,16.71,65.91,-34.56,84.20],[9E9,9E9,9E9,9E9,9E9,9E9]],speeddata0,DefaultBlend,tool0;
  MoveAbsJ [[-19.20,6.94,16.72,66.90,-33.92,84.27],[9E9,9E9,9E9,9E9,9E9,9E9]],speeddata0,DefaultBlend,tool0;
  MoveAbsJ [[-18.96,6.93,16.73,67.89,-33.28,84.34],[9E9,9E9,9E9,9E9,9E9,9E9]],speeddata0,DefaultBlend,tool0;
  MoveAbsJ [[-18.72,6.91,16.75,68.89,-32.65,84.40],[9E9,9E9,9E9,9E9,9E9,9E9]],speeddata0,DefaultBlend,tool0;
  MoveAbsJ [[-18.48,6.89,16.76,69.88,-32.01,84.47],[9E9,9E9,9E9,9E9,9E9,9E9]],speeddata0,DefaultBlend,tool0;
  MoveAbsJ [[-18.24,6.87,16.77,70.87,-31.37,84.54],[9E9,9E9,9E9,9E9,9E9,9E9]],speeddata0,DefaultBlend,tool0;
  MoveAbsJ [[-18.01,6.85,16.78,71.86,-30.74,84.60],[9E9,9E9,9E9,9E9,9E9,9E9]],speeddata0,DefaultBlend,tool0;
  MoveAbsJ [[-17.77,6.83,16.79,72.86,-30.10,84.67],[9E9,9E9,9E9,9E9,9E9,9E9]],speeddata0,DefaultBlend,tool0;
  MoveAbsJ [[-17.53,6.82,16.81,73.85,-29.46,84.74],[9E9,9E9,9E9,9E9,9E9,9E9]],speeddata0,DefaultBlend,tool0;
  MoveAbsJ [[-17.29,6.80,16.82,74.84,-28.83,84.80],[9E9,9E9,9E9,9E9,9E9,9E9]],speeddata0,DefaultBlend,tool0;
  MoveAbsJ [[-17.05,6.78,16.83,75.83,-28.19,84.87],[9E9,9E9,9E9,9E9,9E9,9E9]],speeddata0,DefaultBlend,tool0;
  MoveAbsJ [[-16.81,6.76,16.84,76.82,-27.55,84.94],[9E9,9E9,9E9,9E9,9E9,9E9]],speeddata0,DefaultBlend,tool0;
  MoveAbsJ [[-16.57,6.74,16.85,77.82,-26.92,85.00],[9E9,9E9,9E9,9E9,9E9,9E9]],speeddata0,DefaultBlend,tool0;
  MoveAbsJ [[-16.34,6.73,16.87,78.81,-26.28,85.07],[9E9,9E9,9E9,9E9,9E9,9E9]],speeddata0,DefaultBlend,tool0;
  MoveAbsJ [[-16.10,6.71,16.88,79.80,-25.65,85.14],[9E9,9E9,9E9,9E9,9E9,9E9]],speeddata0,DefaultBlend,tool0;
  MoveAbsJ [[-15.86,6.69,16.89,80.79,-25.01,85.20],[9E9,9E9,9E9,9E9,9E9,9E9]],speeddata0,DefaultBlend,tool0;
  MoveAbsJ [[-15.62,6.67,16.90,81.79,-24.37,85.27],[9E9,9E9,9E9,9E9,9E9,9E9]],speeddata0,DefaultBlend,tool0;
  MoveAbsJ [[-15.38,6.65,16.91,82.78,-23.74,85.34],[9E9,9E9,9E9,9E9,9E9,9E9]],speeddata0,DefaultBlend,tool0;
  MoveAbsJ [[-15.14,6.63,16.92,83.77,-23.10,85.40],[9E9,9E9,9E9,9E9,9E9,9E9]],speeddata0,DefaultBlend,tool0;
  MoveAbsJ [[-14.91,6.62,16.94,84.76,-22.46,85.47],[9E9,9E9,9E9,9E9,9E9,9E9]],speeddata0,DefaultBlend,tool0;
  MoveAbsJ [[-14.67,6.60,16.95,85.75,-21.83,85.54],[9E9,9E9,9E9,9E9,9E9,9E9]],speeddata0,DefaultBlend,tool0;
  MoveAbsJ [[-14.43,6.58,16.96,86.75,-21.19,85.60],[9E9,9E9,9E9,9E9,9E9,9E9]],speeddata0,DefaultBlend,tool0;
  MoveAbsJ [[-14.19,6.56,16.97,87.74,-20.55,85.67],[9E9,9E9,9E9,9E9,9E9,9E9]],speeddata0,DefaultBlend,tool0;
  MoveAbsJ [[-13.95,6.54,16.98,88.73,-19.92,85.73],[9E9,9E9,9E9,9E9,9E9,9E9]],speeddata0,DefaultBlend,tool0;
  MoveAbsJ [[-13.71,6.52,17.00,89.72,-19.28,85.80],[9E9,9E9,9E9,9E9,9E9,9E9]],speeddata0,DefaultBlend,tool0;
  MoveAbsJ [[-13.48,6.51,17.01,90.72,-18.64,85.87],[9E9,9E9,9E9,9E9,9E9,9E9]],speeddata0,DefaultBlend,tool0;
  MoveAbsJ [[-13.24,6.49,17.02,91.71,-18.01,85.93],[9E9,9E9,9E9,9E9,9E9,9E9]],speeddata0,DefaultBlend,tool0;
  MoveAbsJ [[-13.00,6.47,17.03,92.70,-17.37,86.00],[9E9,9E9,9E9,9E9,9E9,9E9]],speeddata0,DefaultBlend,tool0;
  MoveAbsJ [[-12.76,6.45,17.04,93.69,-16.74,86.07],[9E9,9E9,9E9,9E9,9E9,9E9]],speeddata0,DefaultBlend,tool0;
  MoveAbsJ [[-12.52,6.43,17.06,94.68,-16.10,86.13],[9E9,9E9,9E9,9E9,9E9,9E9]],speeddata0,DefaultBlend,tool0;
  MoveAbsJ [[-12.28,6.41,17.07,95.68,-15.46,86.20],[9E9,9E9,9E9,9E9,9E9,9E9]],speeddata0,DefaultBlend,tool0;
  MoveAbsJ [[-12.04,6.40,17.08,96.67,-14.83,86.27],[9E9,9E9,9E9,9E9,9E9,9E9]],speeddata0,DefaultBlend,tool0;
  MoveAbsJ [[-11.81,6.38,17.09,97.66,-14.19,86.33],[9E9,9E9,9E9,9E9,9E9,9E9]],speeddata0,DefaultBlend,tool0;
  MoveAbsJ [[-11.57,6.36,17.10,98.65,-13.55,86.40],[9E9,9E9,9E9,9E9,9E9,9E9]],speeddata0,DefaultBlend,tool0;
  MoveAbsJ [[-11.33,6.34,17.12,99.64,-12.92,86.47],[9E9,9E9,9E9,9E9,9E9,9E9]],speeddata0,DefaultBlend,tool0;
  MoveAbsJ [[-11.09,6.32,17.13,100.64,-12.28,86.53],[9E9,9E9,9E9,9E9,9E9,9E9]],speeddata0,DefaultBlend,tool0;
  MoveAbsJ [[-10.85,6.31,17.14,101.63,-11.64,86.60],[9E9,9E9,9E9,9E9,9E9,9E9]],speeddata0,DefaultBlend,tool0;
  MoveAbsJ [[-10.61,6.29,17.15,102.62,-11.01,86.67],[9E9,9E9,9E9,9E9,9E9,9E9]],speeddata0,DefaultBlend,tool0;
  MoveAbsJ [[-10.38,6.27,17.16,103.61,-10.37,86.73],[9E9,9E9,9E9,9E9,9E9,9E9]],speeddata0,DefaultBlend,tool0;
  MoveAbsJ [[-10.14,6.25,17.18,104.61,-9.73,86.80],[9E9,9E9,9E9,9E9,9E9,9E9]],speeddata0,DefaultBlend,tool0;
  MoveAbsJ [[-9.90,6.23,17.19,105.60,-9.10,86.87],[9E9,9E9,9E9,9E9,9E9,9E9]],speeddata0,DefaultBlend,tool0;
  MoveAbsJ [[-9.66,6.21,17.20,106.59,-8.46,86.93],[9E9,9E9,9E9,9E9,9E9,9E9]],speeddata0,DefaultBlend,tool0;
  MoveAbsJ [[-9.42,6.20,17.21,107.58,-7.82,87.00],[9E9,9E9,9E9,9E9,9E9,9E9]],speeddata0,DefaultBlend,tool0;
  MoveAbsJ [[-9.18,6.18,17.22,108.57,-7.19,87.07],[9E9,9E9,9E9,9E9,9E9,9E9]],speeddata0,DefaultBlend,tool0;
  MoveAbsJ [[-8.95,6.16,17.24,109.57,-6.55,87.13],[9E9,9E9,9E9,9E9,9E9,9E9]],speeddata0,DefaultBlend,tool0;
  MoveAbsJ [[-8.71,6.14,17.25,110.56,-5.92,87.20],[9E9,9E9,9E9,9E9,9E9,9E9]],speeddata0,DefaultBlend,tool0;
  MoveAbsJ [[-8.47,6.12,17.26,111.55,-5.28,87.27],[9E9,9E9,9E9,9E9,9E9,9E9]],speeddata0,DefaultBlend,tool0;
  MoveAbsJ [[-8.23,6.10,17.27,112.54,-4.64,87.33],[9E9,9E9,9E9,9E9,9E9,9E9]],speeddata0,DefaultBlend,tool0;
  MoveAbsJ [[-7.99,6.09,17.28,113.54,-4.01,87.40],[9E9,9E9,9E9,9E9,9E9,9E9]],speeddata0,DefaultBlend,tool0;
  MoveAbsJ [[-7.75,6.07,17.30,114.53,-3.37,87.47],[9E9,9E9,9E9,9E9,9E9,9E9]],speeddata0,DefaultBlend,tool0;
  MoveAbsJ [[-7.51,6.05,17.31,115.52,-2.73,87.53],[9E9,9E9,9E9,9E9,9E9,9E9]],speeddata0,DefaultBlend,tool0;
  MoveAbsJ [[-7.28,6.03,17.32,116.51,-2.10,87.60],[9E9,9E9,9E9,9E9,9E9,9E9]],speeddata0,DefaultBlend,tool0;
  MoveAbsJ [[-7.04,6.01,17.33,117.50,-1.46,87.67],[9E9,9E9,9E9,9E9,9E9,9E9]],speeddata0,DefaultBlend,tool0;
  MoveAbsJ [[-6.80,6.00,17.34,118.50,-0.82,87.73],[9E9,9E9,9E9,9E9,9E9,9E9]],speeddata0,DefaultBlend,tool0;
  MoveAbsJ [[-6.56,5.98,17.36,119.49,-0.19,87.80],[9E9,9E9,9E9,9E9,9E9,9E9]],speeddata0,DefaultBlend,tool0;
  MoveAbsJ [[-6.32,5.96,17.37,120.48,0.45,87.87],[9E9,9E9,9E9,9E9,9E9,9E9]],speeddata0,DefaultBlend,tool0;
  MoveAbsJ [[-6.08,5.94,17.38,121.47,1.09,87.93],[9E9,9E9,9E9,9E9,9E9,9E9]],speeddata0,DefaultBlend,tool0;
  MoveAbsJ [[-5.85,5.92,17.39,122.47,1.72,88.00],[9E9,9E9,9E9,9E9,9E9,9E9]],speeddata0,DefaultBlend,tool0;
  MoveAbsJ [[-5.61,5.90,17.40,123.46,2.36,88.07],[9E9,9E9,9E9,9E9,9E9,9E9]],speeddata0,DefaultBlend,tool0;
  MoveAbsJ [[-5.37,5.89,17.42,124.45,2.99,88.13],[9E9,9E9,9E9,9E9,9E9,9E9]],speeddata0,DefaultBlend,tool0;
  MoveAbsJ [[-5.13,5.87,17.43,125.44,3.63,88.20],[9E9,9E9,9E9,9E9,9E9,9E9]],speeddata0,DefaultBlend,tool0;
  MoveAbsJ [[-4.89,5.85,17.44,126.43,4.27,88.27],[9E9,9E9,9E9,9E9,9E9,9E9]],speeddata0,DefaultBlend,tool0;
  MoveAbsJ [[-4.65,5.83,17.45,127.43,4.90,88.33],[9E9,9E9,9E9,9E9,9E9,9E9]],speeddata0,DefaultBlend,tool0;
  MoveAbsJ [[-4.42,5.81,17.46,128.42,5.54,88.40],[9E9,9E9,9E9,9E9,9E9,9E9]],speeddata0,DefaultBlend,tool0;
  MoveAbsJ [[-4.18,5.79,17.48,129.41,6.18,88.47],[9E9,9E9,9E9,9E9,9E9,9E9]],speeddata0,DefaultBlend,tool0;
  MoveAbsJ [[-3.94,5.78,17.49,130.40,6.81,88.53],[9E9,9E9,9E9,9E9,9E9,9E9]],speeddata0,DefaultBlend,tool0;
  MoveAbsJ [[-3.70,5.76,17.50,131.40,7.45,88.60],[9E9,9E9,9E9,9E9,9E9,9E9]],speeddata0,DefaultBlend,tool0;
  MoveAbsJ [[-3.46,5.74,17.51,132.39,8.09,88.67],[9E9,9E9,9E9,9E9,9E9,9E9]],speeddata0,DefaultBlend,tool0;
  MoveAbsJ [[-3.22,5.72,17.52,133.38,8.72,88.73],[9E9,9E9,9E9,9E9,9E9,9E9]],speeddata0,DefaultBlend,tool0;
  MoveAbsJ [[-2.98,5.70,17.54,134.37,9.36,88.80],[9E9,9E9,9E9,9E9,9E9,9E9]],speeddata0,DefaultBlend,tool0;
  MoveAbsJ [[-2.75,5.68,17.55,135.36,10.00,88.87],[9E9,9E9,9E9,9E9,9E9,9E9]],speeddata0,DefaultBlend,tool0;
  MoveAbsJ [[-2.51,5.67,17.56,136.36,10.63,88.93],[9E9,9E9,9E9,9E9,9E9,9E9]],speeddata0,DefaultBlend,tool0;
  MoveAbsJ [[-2.27,5.65,17.57,137.35,11.27,89.00],[9E9,9E9,9E9,9E9,9E9,9E9]],speeddata0,DefaultBlend,tool0;
  MoveAbsJ [[-2.03,5.63,17.58,138.34,11.91,89.07],[9E9,9E9,9E9,9E9,9E9,9E9]],speeddata0,DefaultBlend,tool0;
  MoveAbsJ [[-1.79,5.61,17.60,139.33,12.54,89.13],[9E9,9E9,9E9,9E9,9E9,9E9]],speeddata0,DefaultBlend,tool0;
  MoveAbsJ [[-1.55,5.59,17.61,140.32,13.18,89.20],[9E9,9E9,9E9,9E9,9E9,9E9]],speeddata0,DefaultBlend,tool0;
  MoveAbsJ [[-1.32,5.58,17.62,141.32,13.81,89.27],[9E9,9E9,9E9,9E9,9E9,9E9]],speeddata0,DefaultBlend,tool0;
  MoveAbsJ [[-1.08,5.56,17.63,142.31,14.45,89.33],[9E9,9E9,9E9,9E9,9E9,9E9]],speeddata0,DefaultBlend,tool0;
  MoveAbsJ [[-0.84,5.54,17.64,143.30,15.09,89.40],[9E9,9E9,9E9,9E9,9E9,9E9]],speeddata0,DefaultBlend,tool0;
  MoveAbsJ [[-0.60,5.52,17.66,144.29,15.72,89.47],[9E9,9E9,9E9,9E9,9E9,9E9]],speeddata0,DefaultBlend,tool0;
  MoveAbsJ [[-0.36,5.50,17.67,145.29,16.36,89.53],[9E9,9E9,9E9,9E9,9E9,9E9]],speeddata0,DefaultBlend,tool0;
  MoveAbsJ [[-0.12,5.48,17.68,146.28,17.00,89.60],[9E9,9E9,9E9,9E9,9E9,9E9]],speeddata0,DefaultBlend,tool0;
  MoveAbsJ [[0.12,5.47,17.69,147.27,17.63,89.67],[9E9,9E9,9E9,9E9,9E9,9E9]],speeddata0,DefaultBlend,tool0;
  MoveAbsJ [[0.35,5.45,17.70,148.26,18.27,89.73],[9E9,9E9,9E9,9E9,9E9,9E9]],speeddata0,DefaultBlend,tool0;
  MoveAbsJ [[0.59,5.43,17.72,149.25,18.91,89.80],[9E9,9E9,9E9,9E9,9E9,9E9]],speeddata0,DefaultBlend,tool0;
  MoveAbsJ [[0.83,5.41,17.73,150.25,19.54,89.86],[9E9,9E9,9E9,9E9,9E9,9E9]],speeddata0,DefaultBlend,tool0;
  MoveAbsJ [[1.07,5.39,17.74,151.24,20.18,89.93],[9E9,9E9,9E9,9E9,9E9,9E9]],speeddata0,DefaultBlend,tool0;
  MoveAbsJ [[1.31,5.37,17.75,152.23,20.82,90.00],[9E9,9E9,9E9,9E9,9E9,9E9]],speeddata0,DefaultBlend,tool0;
  MoveAbsJ [[1.55,5.36,17.76,153.22,21.45,90.06],[9E9,9E9,9E9,9E9,9E9,9E9]],speeddata0,DefaultBlend,tool0;
  MoveAbsJ [[1.78,5.34,17.78,154.22,22.09,90.13],[9E9,9E9,9E9,9E9,9E9,9E9]],speeddata0,DefaultBlend,tool0;
  MoveAbsJ [[2.02,5.32,17.79,155.21,22.72,90.20],[9E9,9E9,9E9,9E9,9E9,9E9]],speeddata0,DefaultBlend,tool0;
  MoveAbsJ [[1.94,5.49,18.06,156.20,23.18,90.19],[9E9,9E9,9E9,9E9,9E9,9E9]],speeddata0,DefaultBlend,tool0;
  MoveAbsJ [[1.86,5.65,18.34,157.19,23.64,90.18],[9E9,9E9,9E9,9E9,9E9,9E9]],speeddata0,DefaultBlend,tool0;
  MoveAbsJ [[1.78,5.82,18.61,158.18,24.10,90.18],[9E9,9E9,9E9,9E9,9E9,9E9]],speeddata0,DefaultBlend,tool0;
